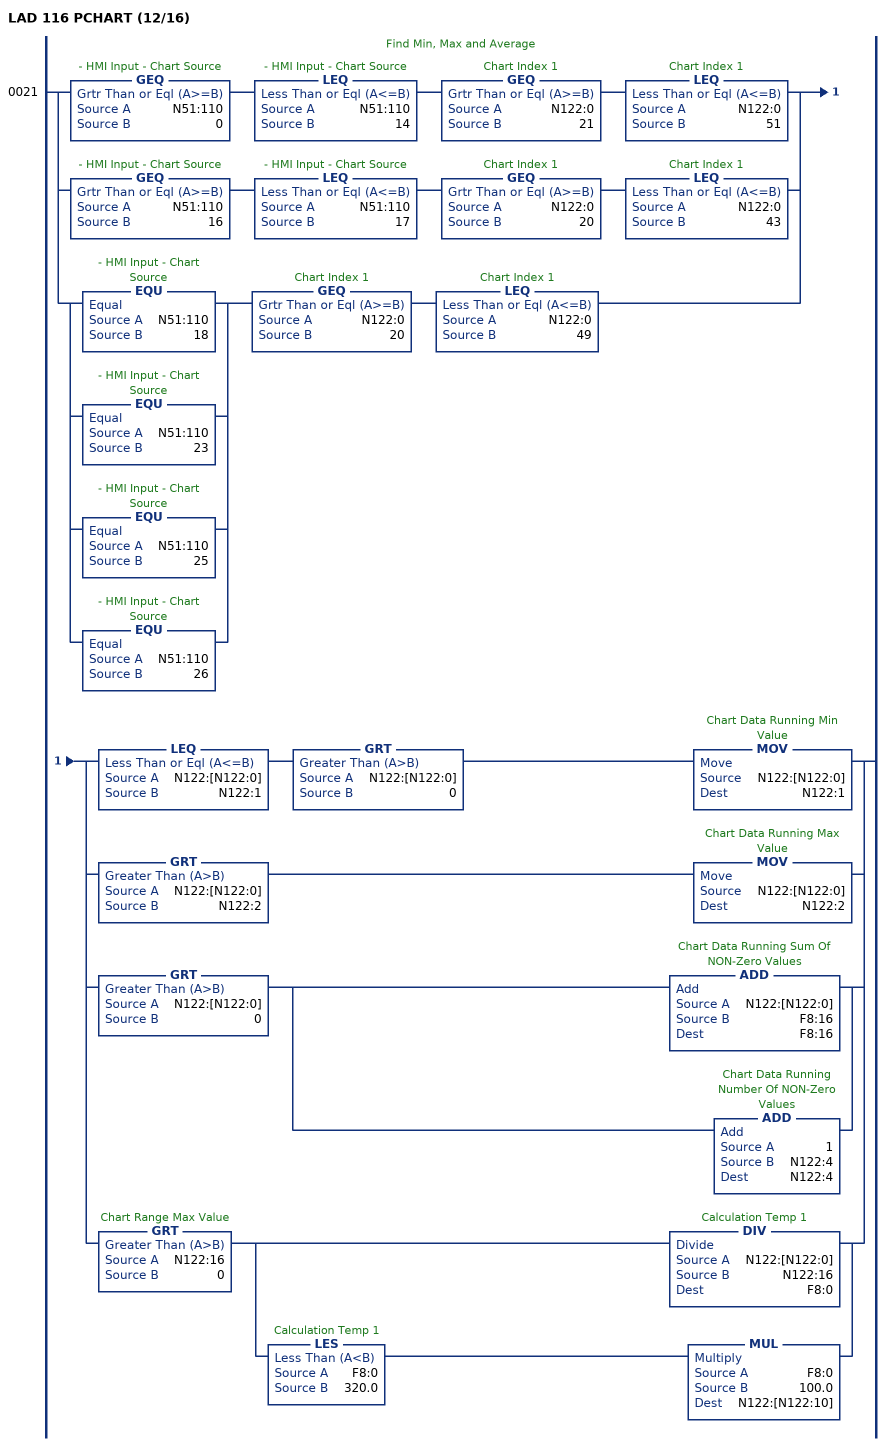
% Rung: 21 %
% Find Min, Max and Average %
SOR BST GEQ N51:110 0 LEQ N51:110 14 GEQ N122:0 21 LEQ N122:0 51 NXB GEQ N51:110 16 LEQ N51:110 17 GEQ N122:0 20 LEQ N122:0 43 NXB BST EQU N51:110 18 NXB EQU N51:110 23 NXB EQU N51:110 25 NXB EQU N51:110 26 BND GEQ N122:0 20 LEQ N122:0 49 BND BST LEQ N122:[N122:0] N122:1 GRT N122:[N122:0] 0 MOV N122:[N122:0] N122:1 NXB GRT N122:[N122:0] N122:2 MOV N122:[N122:0] N122:2 NXB GRT N122:[N122:0] 0 BST ADD N122:[N122:0] F8:16 F8:16 NXB ADD 1 N122:4 N122:4 BND NXB GRT N122:16 0 BST DIV N122:[N122:0] N122:16 F8:0 NXB LES F8:0 320.0 MUL F8:0 100.0 N122:[N122:10] BND BND EOR
%   N51:110  "- HMI Input - Chart Source" %
%   N122:0  "Chart Index 1" %
%   N122:1  "Chart Data Running Min Value" %
%   N122:2  "Chart Data Running Max Value" %
%   F8:16  "Chart Data Running Sum Of NON-Zero Values" %
%   N122:4  "Chart Data Running Number Of NON-Zero Values" %
%   N122:16  "Chart Range Max Value" %
%   F8:0  "Calculation Temp 1" %
%   N122:10  "Chart Index 2" %

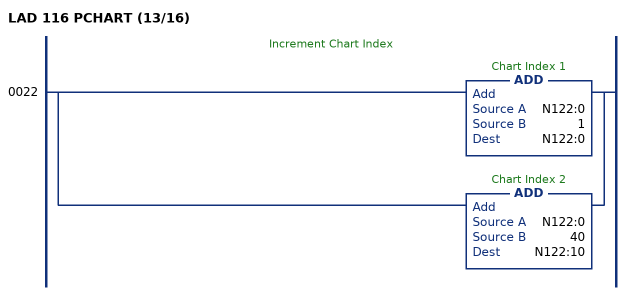
% Rung: 22 %
% Increment Chart Index %
SOR BST ADD N122:0 1 N122:0 NXB ADD N122:0 40 N122:10 BND EOR
%   N122:0  "Chart Index 1" %
%   N122:10  "Chart Index 2" %

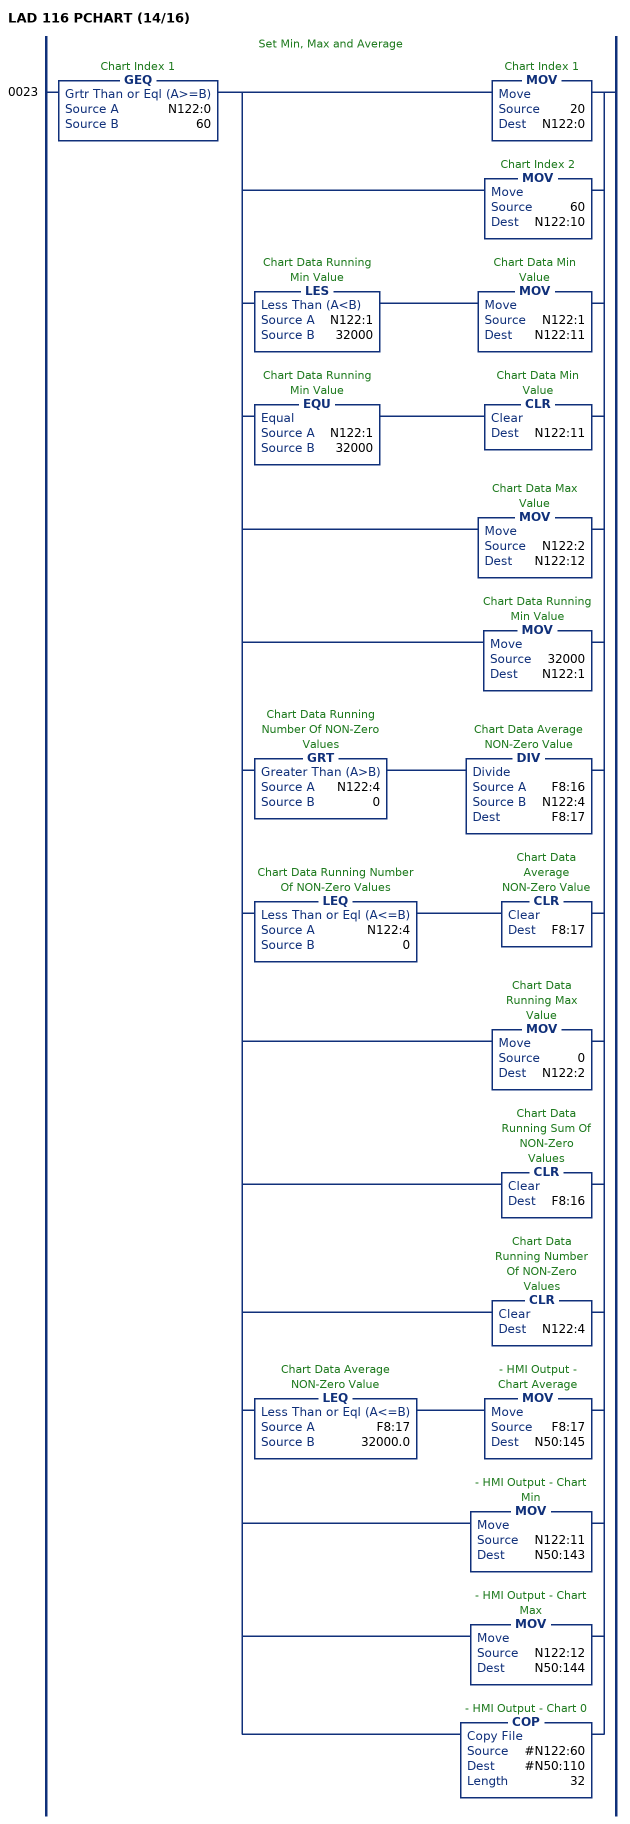
% Rung: 23 %
% Set Min, Max and Average %
SOR GEQ N122:0 60 BST MOV 20 N122:0 NXB MOV 60 N122:10 NXB BST LES N122:1 32000 MOV N122:1 N122:11 NXB EQU N122:1 32000 CLR N122:11 BND NXB MOV N122:2 N122:12 NXB MOV 32000 N122:1 NXB BST GRT N122:4 0 DIV F8:16 N122:4 F8:17 NXB LEQ N122:4 0 CLR F8:17 BND NXB MOV 0 N122:2 NXB CLR F8:16 NXB CLR N122:4 NXB LEQ F8:17 32000.0 MOV F8:17 N50:145 NXB MOV N122:11 N50:143 NXB MOV N122:12 N50:144 NXB COP #N122:60 #N50:110 32 BND EOR
%   N122:0  "Chart Index 1" %
%   N122:10  "Chart Index 2" %
%   N122:1  "Chart Data Running Min Value" %
%   N122:11  "Chart Data Min Value" %
%   N122:2  "Chart Data Running Max Value" %
%   N122:12  "Chart Data Max Value" %
%   N122:4  "Chart Data Running Number Of NON-Zero Values" %
%   F8:16  "Chart Data Running Sum Of NON-Zero Values" %
%   F8:17  "Chart Data Average NON-Zero Value" %
%   N50:145  "- HMI Output - Chart Average" %
%   N50:143  "- HMI Output - Chart Min" %
%   N50:144  "- HMI Output - Chart Max" %
%   N50:110  "- HMI Output - Chart 0" %

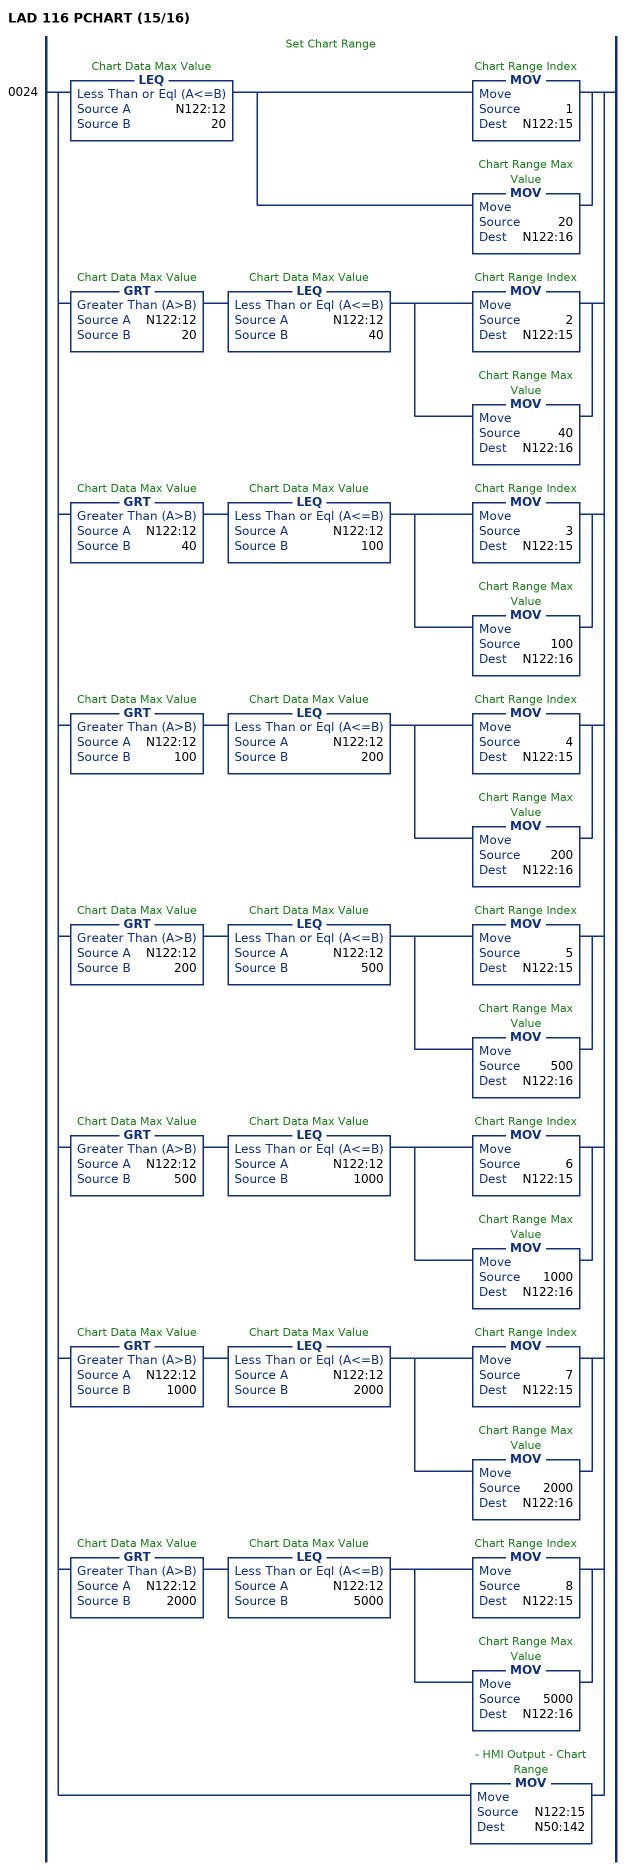
% Rung: 24 %
% Set Chart Range %
SOR BST LEQ N122:12 20 BST MOV 1 N122:15 NXB MOV 20 N122:16 BND NXB GRT N122:12 20 LEQ N122:12 40 BST MOV 2 N122:15 NXB MOV 40 N122:16 BND NXB GRT N122:12 40 LEQ N122:12 100 BST MOV 3 N122:15 NXB MOV 100 N122:16 BND NXB GRT N122:12 100 LEQ N122:12 200 BST MOV 4 N122:15 NXB MOV 200 N122:16 BND NXB GRT N122:12 200 LEQ N122:12 500 BST MOV 5 N122:15 NXB MOV 500 N122:16 BND NXB GRT N122:12 500 LEQ N122:12 1000 BST MOV 6 N122:15 NXB MOV 1000 N122:16 BND NXB GRT N122:12 1000 LEQ N122:12 2000 BST MOV 7 N122:15 NXB MOV 2000 N122:16 BND NXB GRT N122:12 2000 LEQ N122:12 5000 BST MOV 8 N122:15 NXB MOV 5000 N122:16 BND NXB MOV N122:15 N50:142 BND EOR
%   N122:12  "Chart Data Max Value" %
%   N122:15  "Chart Range Index" %
%   N122:16  "Chart Range Max Value" %
%   N50:142  "- HMI Output - Chart Range" %

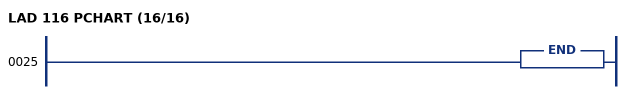
% Rung: 25 %
SOR END EOR

LADDER 117 "CDATA"    % Load Containment Data %
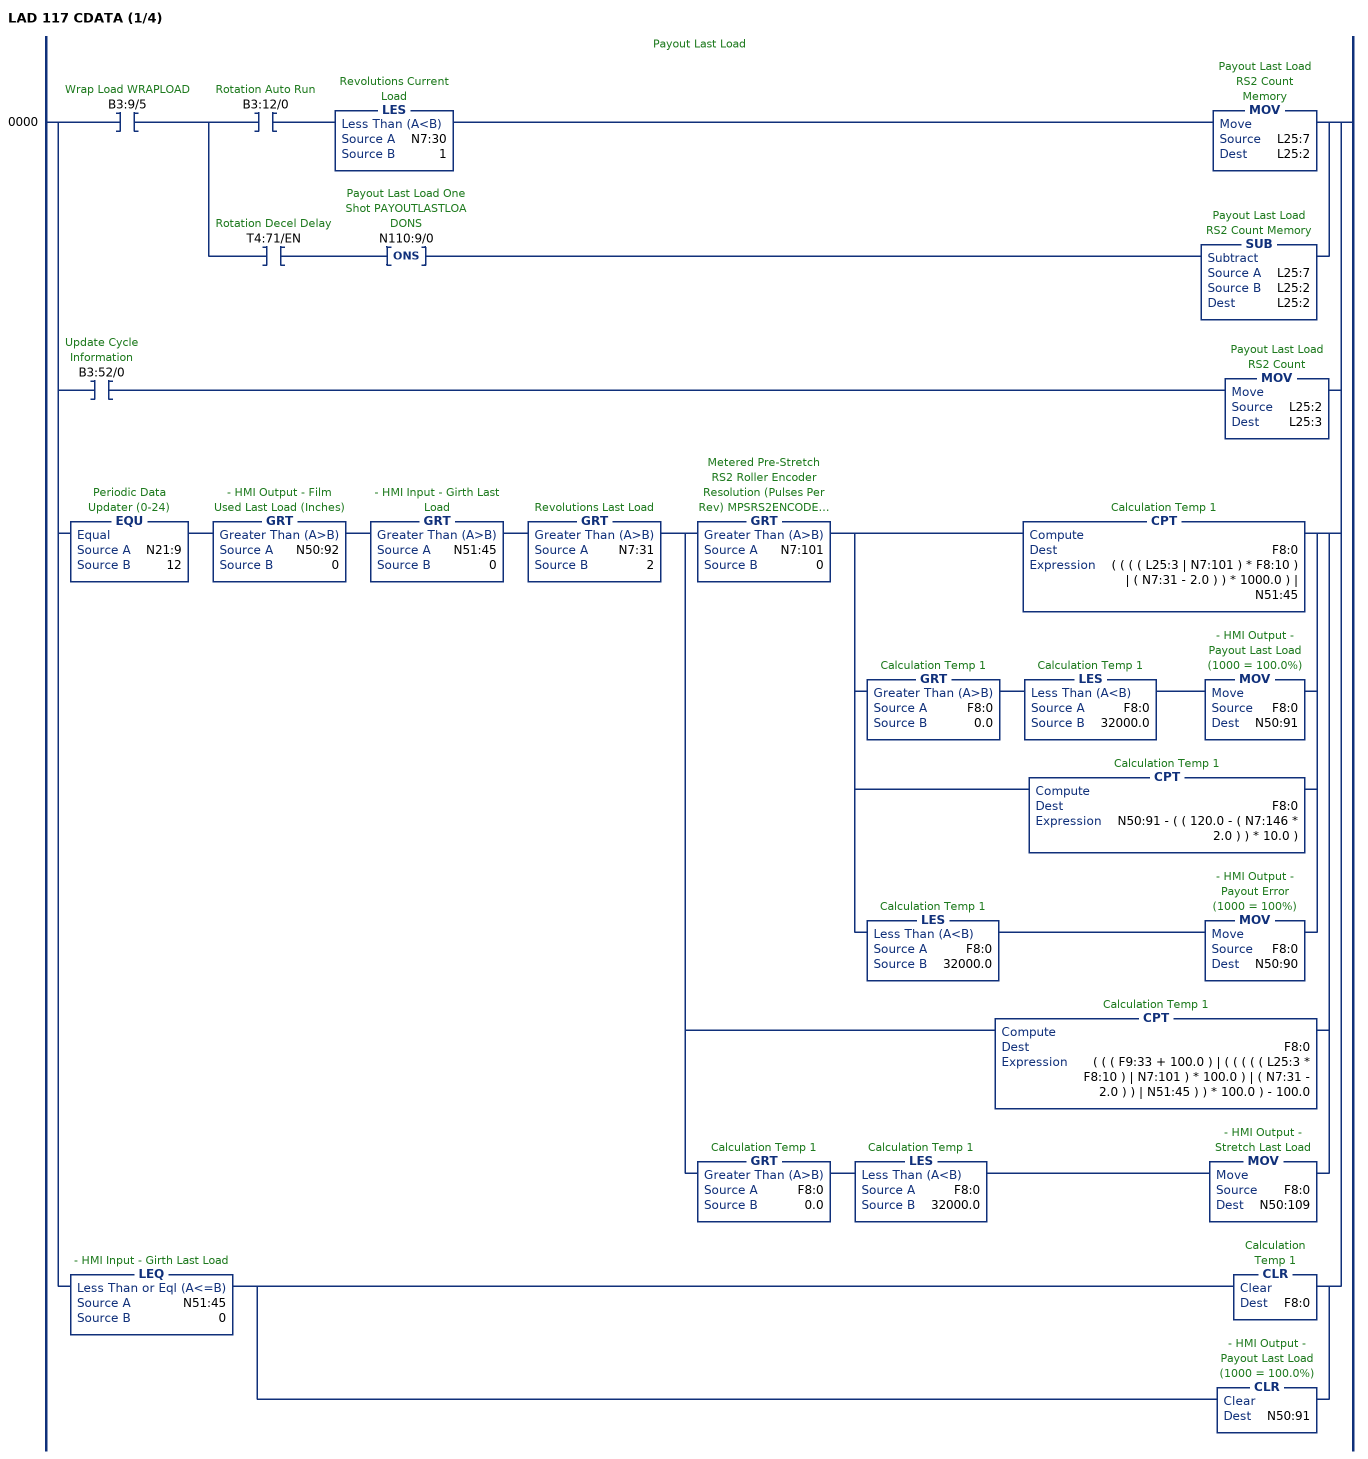
% Rung: 0 %
% Payout Last Load %
SOR BST XIC B3:9/5 BST XIC B3:12/0 LES N7:30 1 MOV L25:7 L25:2 NXB XIC T4:71/EN ONS N110:9/0 SUB L25:7 L25:2 L25:2 BND NXB XIC B3:52/0 MOV L25:2 L25:3 NXB EQU N21:9 12 GRT N50:92 0 GRT N51:45 0 GRT N7:31 2 BST GRT N7:101 0 BST CPT F8:0 " ( ( ( ( L25:3 | N7:101 ) * F8:10 ) | ( N7:31 - 2.0 ) ) * 1000.0 ) | N51:45 " NXB GRT F8:0 0.0 LES F8:0 32000.0 MOV F8:0 N50:91 NXB CPT F8:0 " N50:91 - ( ( 120.0 - ( N7:146 * 2.0 ) ) * 10.0 ) " NXB LES F8:0 32000.0 MOV F8:0 N50:90 BND NXB BST CPT F8:0 " ( ( ( F9:33 + 100.0 ) | ( ( ( ( ( L25:3 * F8:10 ) | N7:101 ) * 100.0 ) | ( N7:31 - 2.0 ) ) | N51:45 ) ) * 100.0 ) - 100.0 " NXB GRT F8:0 0.0 LES F8:0 32000.0 MOV F8:0 N50:109 BND BND NXB LEQ N51:45 0 BST CLR F8:0 NXB CLR N50:91 BND BND EOR
%   B3:9/5  WRAPLOAD  "Wrap Load" %
%   B3:12/0  "Rotation Auto Run" %
%   N7:30  "Revolutions Current Load" %
%   L25:7  "Metered Pre-Stretch RS2 Roller Current Count" %
%   L25:2  "Payout Last Load RS2 Count Memory" %
%   T4:71  "Rotation Decel Delay" %
%   N110:9/0  PAYOUTLASTLOADONS  "Payout Last Load One Shot" %
%   B3:52/0  "Update Cycle Information" %
%   L25:3  "Payout Last Load RS2 Count" %
%   N21:9  "Periodic Data Updater (0-24)" %
%   N50:92  "- HMI Output - Film Used Last Load (Inches)" %
%   N51:45  "- HMI Input - Girth Last Load" %
%   N7:31  "Revolutions Last Load" %
%   N7:101  MPSRS2ENCODERRES  "Metered Pre-Stretch RS2 Roller Encoder Resolution (Pulses Per Rev)" %
%   F8:0  "Calculation Temp 1" %
%   F8:10  MPSRS2CIRC  "Metered Pre-Stretch RS2 Roller Circumference (Inches)" %
%   N50:91  "- HMI Output - Payout Last Load (1000 = 100.0%)" %
%   N7:146  FORCELOADLAST  "Force At Load On Last Load" %
%   N50:90  "- HMI Output - Payout Error (1000 = 100%)" %
%   F9:33  PRESTRETCH  "Pre-Stretch %" %
%   N50:109  "- HMI Output - Stretch Last Load" %

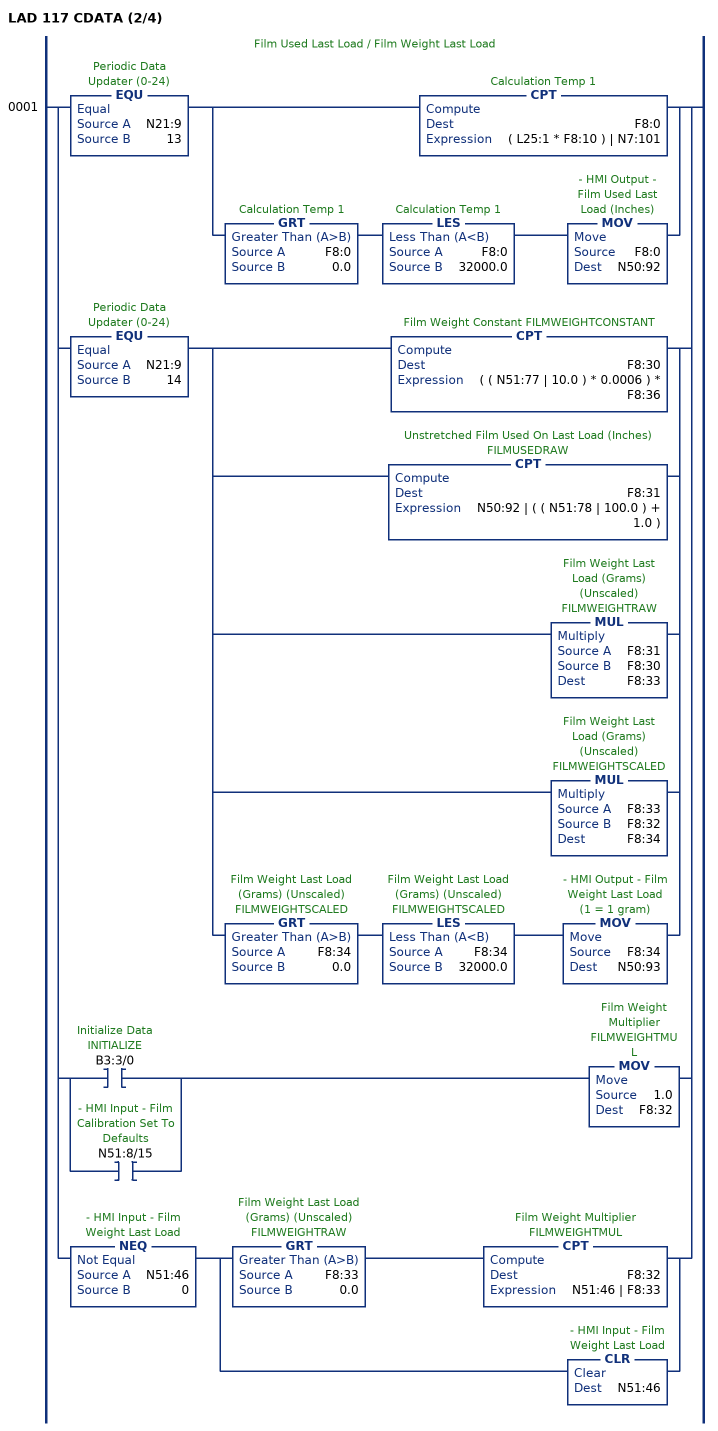
% Rung: 1 %
% Film Used Last Load / Film Weight Last Load %
SOR BST EQU N21:9 13 BST CPT F8:0 " ( L25:1 * F8:10 ) | N7:101 " NXB GRT F8:0 0.0 LES F8:0 32000.0 MOV F8:0 N50:92 BND NXB EQU N21:9 14 BST CPT F8:30 " ( ( N51:77 | 10.0 ) * 0.0006 ) * F8:36 " NXB CPT F8:31 " N50:92 | ( ( N51:78 | 100.0 ) + 1.0 ) " NXB BST MUL F8:31 F8:30 F8:33 NXB MUL F8:33 F8:32 F8:34 NXB GRT F8:34 0.0 LES F8:34 32000.0 MOV F8:34 N50:93 BND BND NXB BST XIC B3:3/0 NXB XIC N51:8/15 BND MOV 1.0 F8:32 NXB NEQ N51:46 0 BST GRT F8:33 0.0 CPT F8:32 " N51:46 | F8:33 " NXB CLR N51:46 BND BND EOR
%   N21:9  "Periodic Data Updater (0-24)" %
%   F8:0  "Calculation Temp 1" %
%   L25:1  "Metered Pre-Stretch RS2 Roller Counts Last Load" %
%   F8:10  MPSRS2CIRC  "Metered Pre-Stretch RS2 Roller Circumference (Inches)" %
%   N7:101  MPSRS2ENCODERRES  "Metered Pre-Stretch RS2 Roller Encoder Resolution (Pulses Per Rev)" %
%   N50:92  "- HMI Output - Film Used Last Load (Inches)" %
%   F8:30  FILMWEIGHTCONSTANT  "Film Weight Constant" %
%   N51:77  "- HMI Input - Preset Film Thickness (in microns)" %
%   F8:36  FILMSIZE  "Film Size (Inches)" %
%   F8:31  FILMUSEDRAW  "Unstretched Film Used On Last Load (Inches)" %
%   N51:78  "- HMI Input - Preset Prestretch %" %
%   F8:33  FILMWEIGHTRAW  "Film Weight Last Load (Grams) (Unscaled)" %
%   F8:32  FILMWEIGHTMUL  "Film Weight Multiplier" %
%   F8:34  FILMWEIGHTSCALED  "Film Weight Last Load (Grams) (Unscaled)" %
%   N50:93  "- HMI Output - Film Weight Last Load (1 = 1 gram)" %
%   B3:3/0  INITIALIZE  "Initialize Data" %
%   N51:8/15  "- HMI Input - Film Calibration Set To Defaults" %
%   N51:46  "- HMI Input - Film Weight Last Load" %

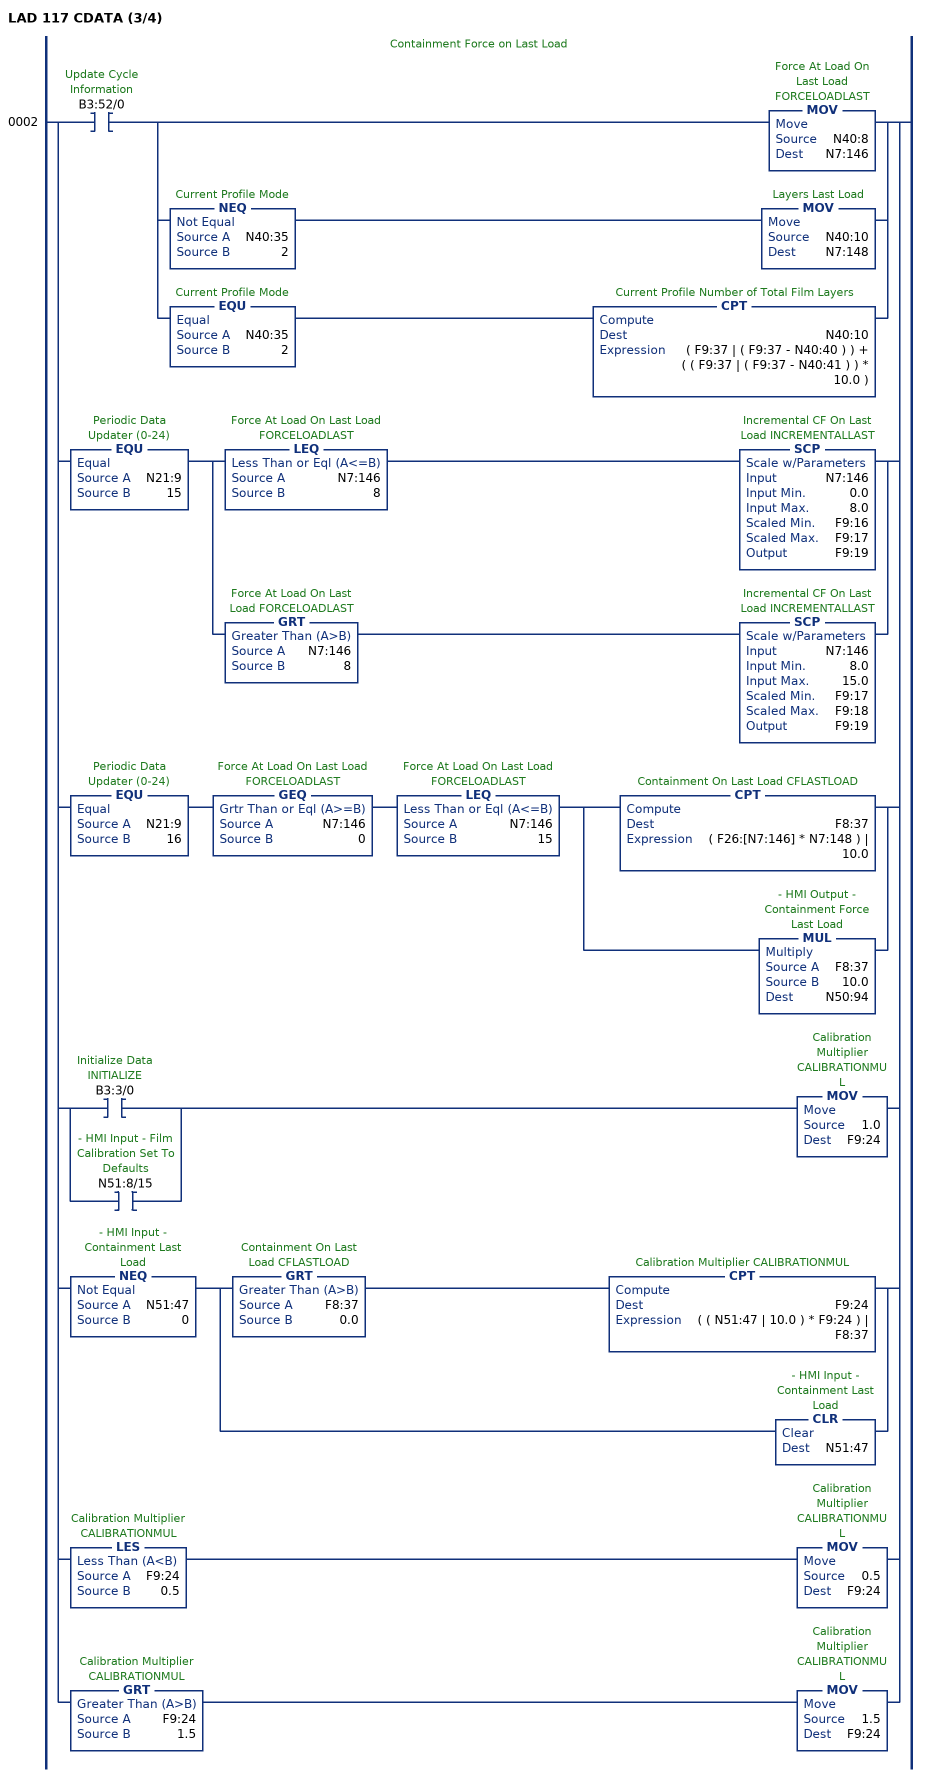
% Rung: 2 %
% Containment Force on Last Load %
SOR BST XIC B3:52/0 BST MOV N40:8 N7:146 NXB NEQ N40:35 2 MOV N40:10 N7:148 NXB EQU N40:35 2 CPT N40:10 " ( F9:37 | ( F9:37 - N40:40 ) ) + ( ( F9:37 | ( F9:37 - N40:41 ) ) * 10.0 ) " BND NXB EQU N21:9 15 BST LEQ N7:146 8 SCP N7:146 0.0 8.0 F9:16 F9:17 F9:19 NXB GRT N7:146 8 SCP N7:146 8.0 15.0 F9:17 F9:18 F9:19 BND NXB EQU N21:9 16 GEQ N7:146 0 LEQ N7:146 15 BST CPT F8:37 " ( F26:[N7:146] * N7:148 ) | 10.0 " NXB MUL F8:37 10.0 N50:94 BND NXB BST XIC B3:3/0 NXB XIC N51:8/15 BND MOV 1.0 F9:24 NXB NEQ N51:47 0 BST GRT F8:37 0.0 CPT F9:24 " ( ( N51:47 | 10.0 ) * F9:24 ) | F8:37 " NXB CLR N51:47 BND NXB LES F9:24 0.5 MOV 0.5 F9:24 NXB GRT F9:24 1.5 MOV 1.5 F9:24 BND EOR
%   B3:52/0  "Update Cycle Information" %
%   N40:8  "Current Profile Force At Load" %
%   N7:146  FORCELOADLAST  "Force At Load On Last Load" %
%   N40:35  "Current Profile Mode" %
%   N40:10  "Current Profile Number of Total Film Layers" %
%   N7:148  "Layers Last Load" %
%   F9:37  "Film Width Scaled for Film Tension" %
%   N21:9  "Periodic Data Updater (0-24)" %
%   F9:16  INCREMENTALAT0  "Incremental CF At WF0 For A Given Film Thickness" %
%   F9:17  INCREMENTALAT8  "Incremental CF At WF8 For A Given Film Thickness" %
%   F9:19  INCREMENTALLAST  "Incremental CF On Last Load" %
%   F9:18  INCREMENTALAT15  "Incremental CF At WF15 For A Given Film Thickness" %
%   F8:37  CFLASTLOAD  "Containment On Last Load" %
%   N50:94  "- HMI Output - Containment Force Last Load" %
%   B3:3/0  INITIALIZE  "Initialize Data" %
%   N51:8/15  "- HMI Input - Film Calibration Set To Defaults" %
%   F9:24  CALIBRATIONMUL  "Calibration Multiplier" %
%   N51:47  "- HMI Input - Containment Last Load" %

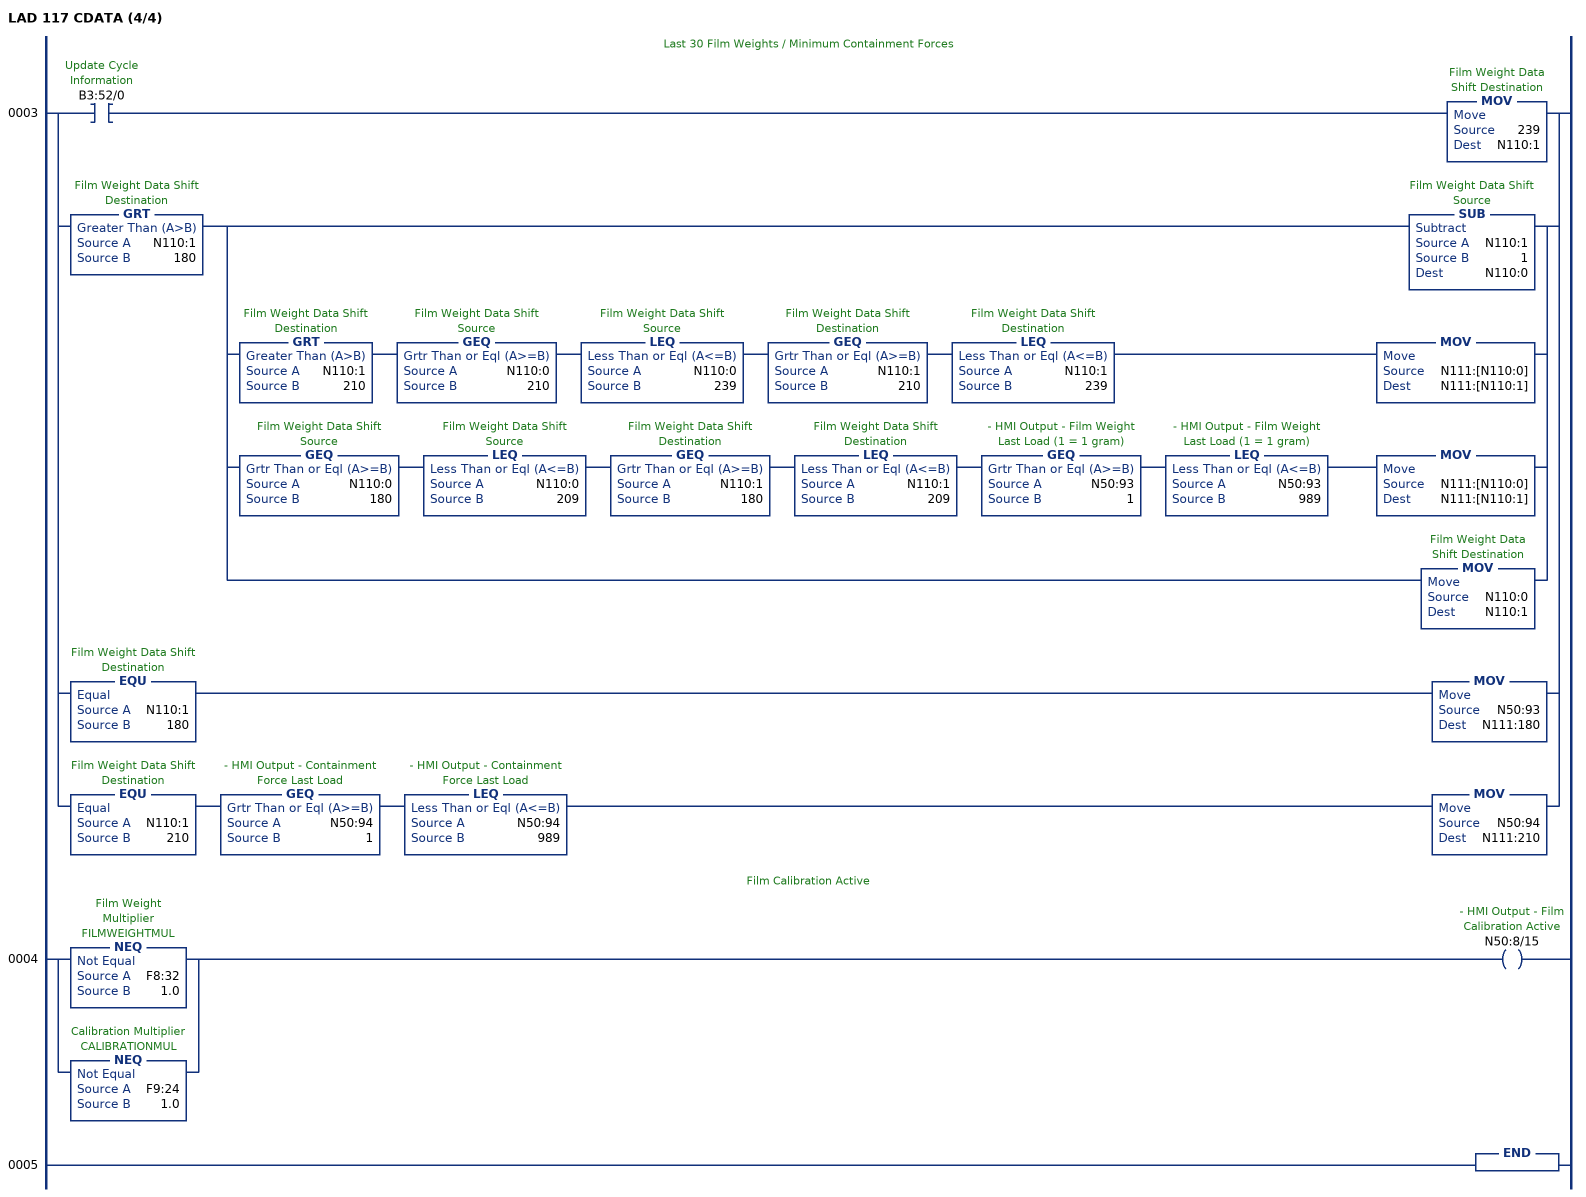
% Rung: 3 %
% Last 30 Film Weights / Minimum Containment Forces %
SOR BST XIC B3:52/0 MOV 239 N110:1 NXB GRT N110:1 180 BST SUB N110:1 1 N110:0 NXB GRT N110:1 210 GEQ N110:0 210 LEQ N110:0 239 GEQ N110:1 210 LEQ N110:1 239 MOV N111:[N110:0] N111:[N110:1] NXB GEQ N110:0 180 LEQ N110:0 209 GEQ N110:1 180 LEQ N110:1 209 GEQ N50:93 1 LEQ N50:93 989 MOV N111:[N110:0] N111:[N110:1] NXB MOV N110:0 N110:1 BND NXB EQU N110:1 180 MOV N50:93 N111:180 NXB EQU N110:1 210 GEQ N50:94 1 LEQ N50:94 989 MOV N50:94 N111:210 BND EOR
%   B3:52/0  "Update Cycle Information" %
%   N110:1  "Film Weight Data Shift Destination" %
%   N110:0  "Film Weight Data Shift Source" %
%   N50:93  "- HMI Output - Film Weight Last Load (1 = 1 gram)" %
%   N50:94  "- HMI Output - Containment Force Last Load" %
% Rung: 4 %
% Film Calibration Active %
SOR BST NEQ F8:32 1.0 NXB NEQ F9:24 1.0 BND OTE N50:8/15 EOR
%   F8:32  FILMWEIGHTMUL  "Film Weight Multiplier" %
%   F9:24  CALIBRATIONMUL  "Calibration Multiplier" %
%   N50:8/15  "- HMI Output - Film Calibration Active" %
% Rung: 5 %
SOR END EOR

LADDER 214 "MPS CALC"
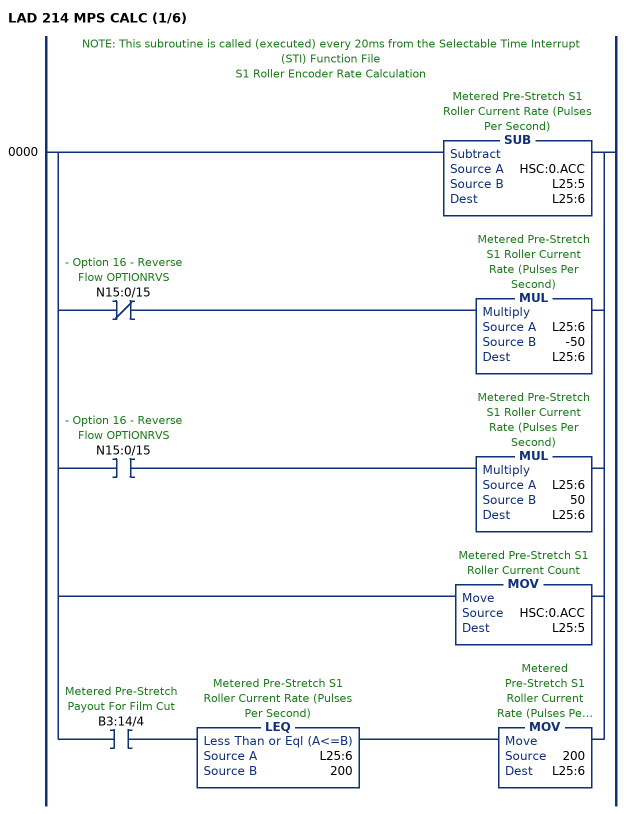
% Rung: 0 %
% NOTE: This subroutine is called (executed) every 20ms from the Selectable Time Interrupt (STI) Function File
% 
% S1 Roller Encoder Rate Calculation %
SOR BST SUB HSC:0.ACC L25:5 L25:6 NXB XIO N15:0/15 MUL L25:6 -50 L25:6 NXB XIC N15:0/15 MUL L25:6 50 L25:6 NXB MOV HSC:0.ACC L25:5 NXB XIC B3:14/4 LEQ L25:6 200 MOV 200 L25:6 BND EOR
%   L25:5  "Metered Pre-Stretch S1 Roller Current Count" %
%   L25:6  "Metered Pre-Stretch S1 Roller Current Rate (Pulses Per Second)" %
%   N15:0/15  OPTIONRVS  "- Option 16 - Reverse Flow" %
%   B3:14/4  "Metered Pre-Stretch Payout For Film Cut" %

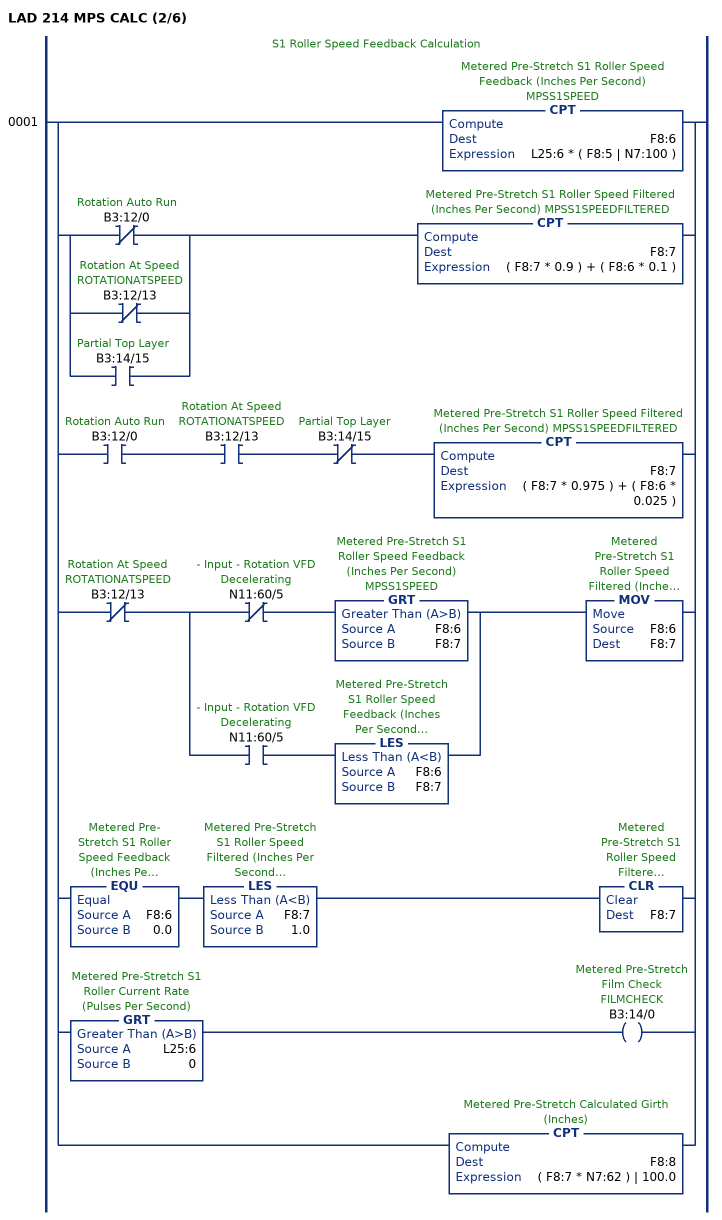
% Rung: 1 %
% S1 Roller Speed Feedback Calculation %
SOR BST CPT F8:6 " L25:6 * ( F8:5 | N7:100 ) " NXB BST XIO B3:12/0 NXB XIO B3:12/13 NXB XIC B3:14/15 BND CPT F8:7 " ( F8:7 * 0.9 ) + ( F8:6 * 0.1 ) " NXB XIC B3:12/0 XIC B3:12/13 XIO B3:14/15 CPT F8:7 " ( F8:7 * 0.975 ) + ( F8:6 * 0.025 ) " NXB XIO B3:12/13 BST XIO N11:60/5 GRT F8:6 F8:7 NXB XIC N11:60/5 LES F8:6 F8:7 BND MOV F8:6 F8:7 NXB EQU F8:6 0.0 LES F8:7 1.0 CLR F8:7 NXB GRT L25:6 0 OTE B3:14/0 NXB CPT F8:8 " ( F8:7 * N7:62 ) | 100.0 " BND EOR
%   F8:6  MPSS1SPEED  "Metered Pre-Stretch S1 Roller Speed Feedback (Inches Per Second)" %
%   L25:6  "Metered Pre-Stretch S1 Roller Current Rate (Pulses Per Second)" %
%   F8:5  MPSS1CIRC  "Metered Pre-Stretch S1 Roller Circumference (Inches)" %
%   N7:100  MPSS1ENCODERRES  "Metered Pre-Stretch S1 Roller Encoder Resolution (Pulses Per Rev)" %
%   B3:12/0  "Rotation Auto Run" %
%   B3:12/13  ROTATIONATSPEED  "Rotation At Speed" %
%   B3:14/15  "Partial Top Layer" %
%   F8:7  MPSS1SPEEDFILTERED  "Metered Pre-Stretch S1 Roller Speed Filtered (Inches Per Second)" %
%   N11:60/5  "- Input - Rotation VFD Decelerating" %
%   B3:14/0  FILMCHECK  "Metered Pre-Stretch Film Check" %
%   F8:8  "Metered Pre-Stretch Calculated Girth (Inches)" %
%   N7:62  "Rotation Revolution Time (100 = 1.00s)" %

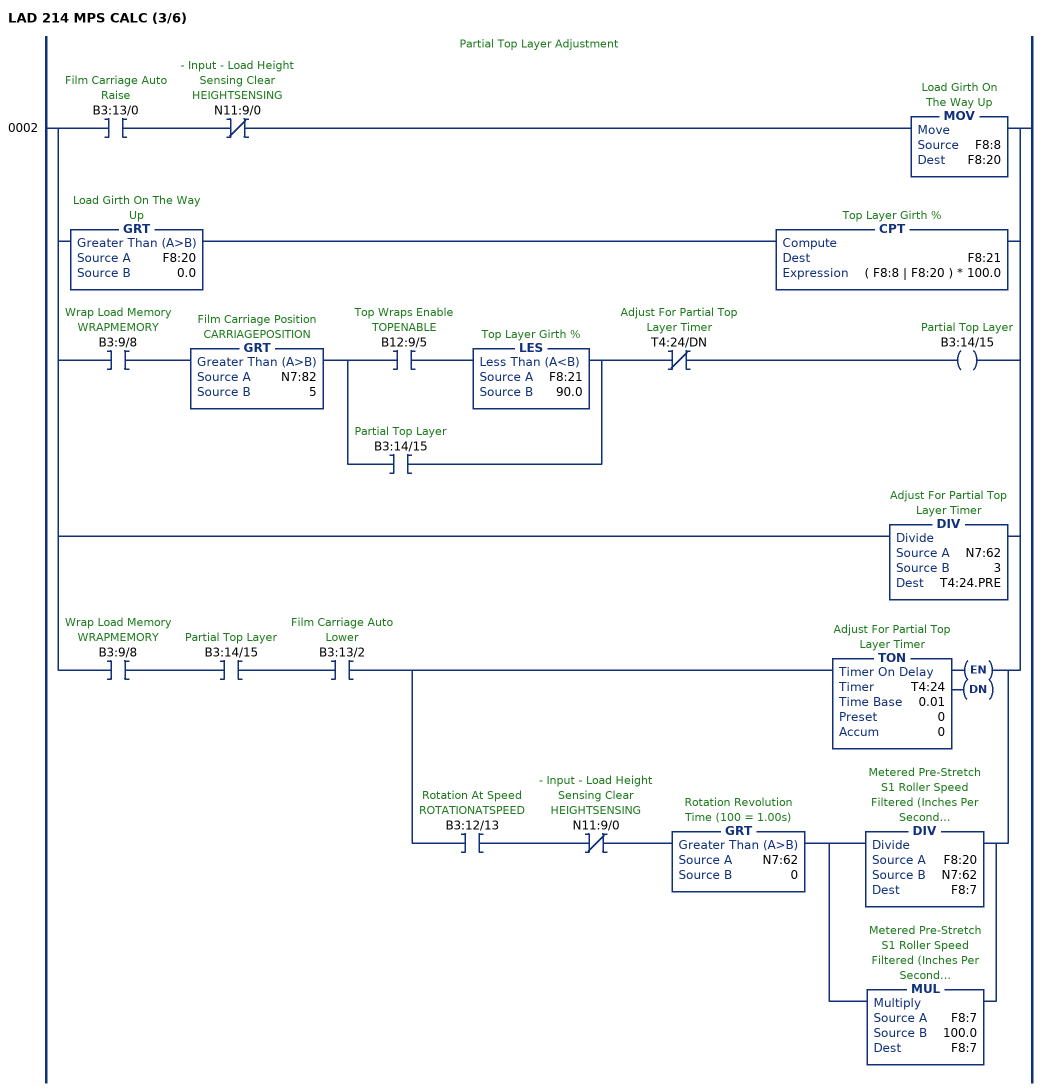
% Rung: 2 %
% Partial Top Layer Adjustment %
SOR BST XIC B3:13/0 XIO N11:9/0 MOV F8:8 F8:20 NXB GRT F8:20 0.0 CPT F8:21 " ( F8:8 | F8:20 ) * 100.0 " NXB XIC B3:9/8 GRT N7:82 5 BST XIC B12:9/5 LES F8:21 90.0 NXB XIC B3:14/15 BND XIO T4:24/DN OTE B3:14/15 NXB DIV N7:62 3 T4:24.PRE NXB XIC B3:9/8 XIC B3:14/15 XIC B3:13/2 BST TON T4:24 0.01 0 0 NXB XIC B3:12/13 XIO N11:9/0 GRT N7:62 0 BST DIV F8:20 N7:62 F8:7 NXB MUL F8:7 100.0 F8:7 BND BND BND EOR
%   B3:13/0  "Film Carriage Auto Raise" %
%   N11:9/0  HEIGHTSENSING  "- Input - Load Height Sensing Clear" %
%   F8:8  "Metered Pre-Stretch Calculated Girth (Inches)" %
%   F8:20  "Load Girth On The Way Up" %
%   F8:21  "Top Layer Girth %" %
%   B3:9/8  WRAPMEMORY  "Wrap Load Memory" %
%   N7:82  CARRIAGEPOSITION  "Film Carriage Position" %
%   B12:9/5  TOPENABLE  "Top Wraps Enable" %
%   B3:14/15  "Partial Top Layer" %
%   T4:24  "Adjust For Partial Top Layer Timer" %
%   N7:62  "Rotation Revolution Time (100 = 1.00s)" %
%   B3:13/2  "Film Carriage Auto Lower" %
%   B3:12/13  ROTATIONATSPEED  "Rotation At Speed" %
%   F8:7  MPSS1SPEEDFILTERED  "Metered Pre-Stretch S1 Roller Speed Filtered (Inches Per Second)" %

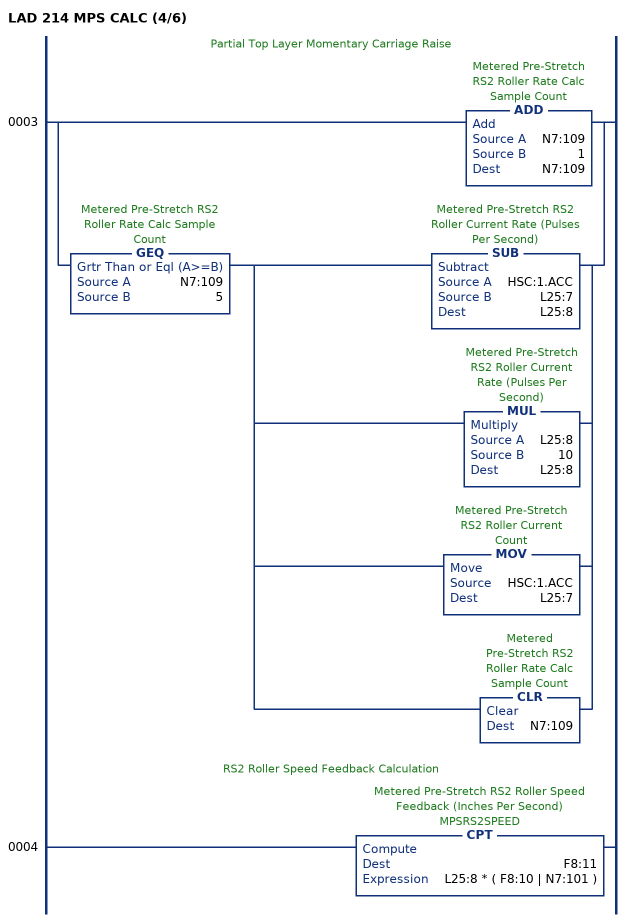
% Rung: 3 %
% Partial Top Layer Momentary Carriage Raise %
SOR BST ADD N7:109 1 N7:109 NXB GEQ N7:109 5 BST SUB HSC:1.ACC L25:7 L25:8 NXB MUL L25:8 10 L25:8 NXB MOV HSC:1.ACC L25:7 NXB CLR N7:109 BND BND EOR
%   N7:109  "Metered Pre-Stretch RS2 Roller Rate Calc Sample Count" %
%   L25:7  "Metered Pre-Stretch RS2 Roller Current Count" %
%   L25:8  "Metered Pre-Stretch RS2 Roller Current Rate (Pulses Per Second)" %
% Rung: 4 %
% RS2 Roller Speed Feedback Calculation %
SOR CPT F8:11 " L25:8 * ( F8:10 | N7:101 ) " EOR
%   F8:11  MPSRS2SPEED  "Metered Pre-Stretch RS2 Roller Speed Feedback (Inches Per Second)" %
%   L25:8  "Metered Pre-Stretch RS2 Roller Current Rate (Pulses Per Second)" %
%   F8:10  MPSRS2CIRC  "Metered Pre-Stretch RS2 Roller Circumference (Inches)" %
%   N7:101  MPSRS2ENCODERRES  "Metered Pre-Stretch RS2 Roller Encoder Resolution (Pulses Per Rev)" %

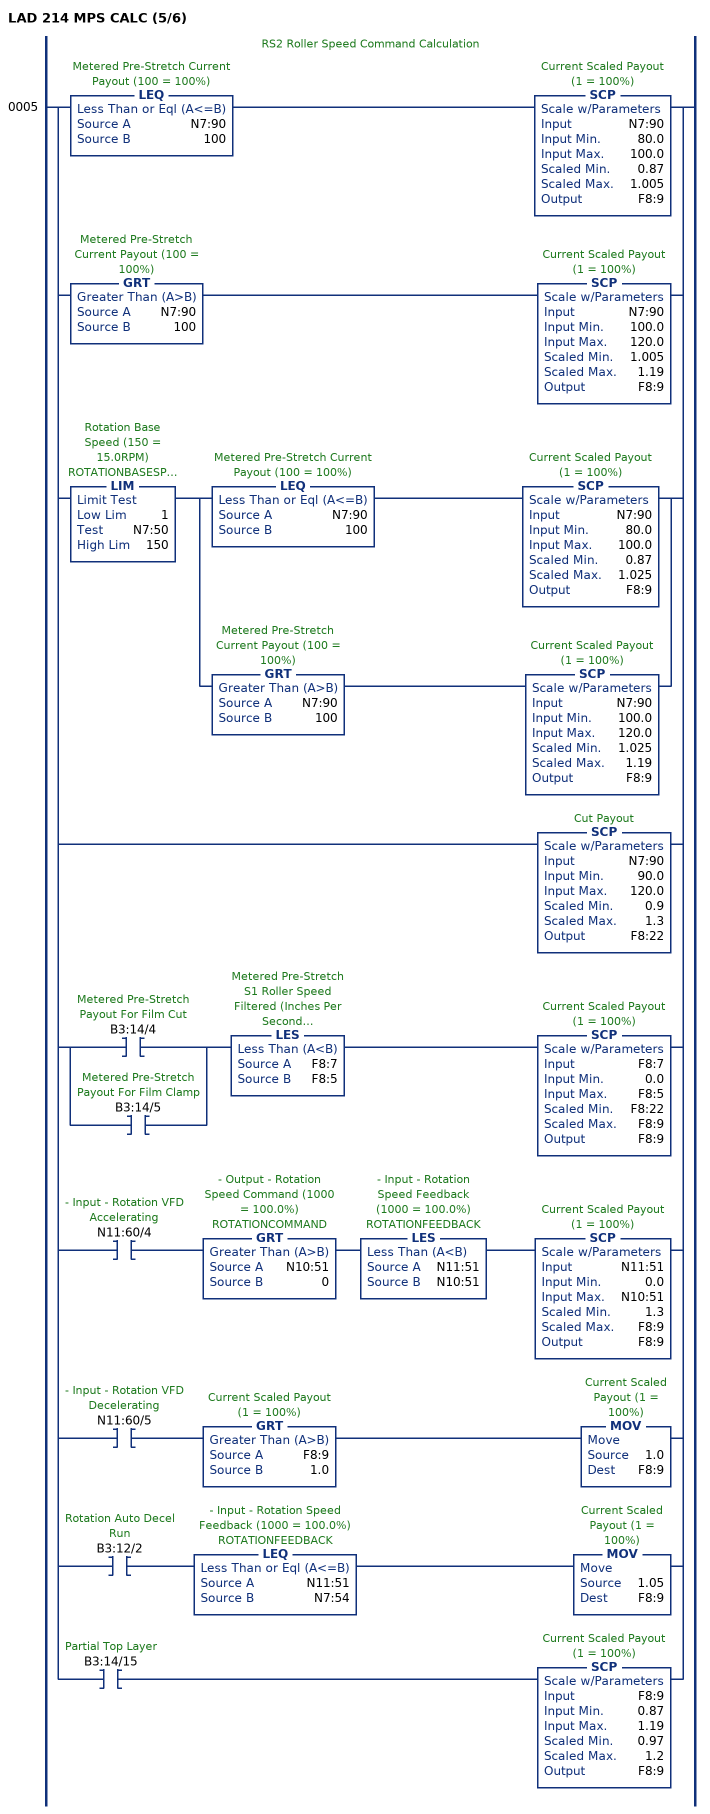
% Rung: 5 %
% RS2 Roller Speed Command Calculation %
SOR BST BST LEQ N7:90 100 SCP N7:90 80.0 100.0 0.87 1.005 F8:9 NXB GRT N7:90 100 SCP N7:90 100.0 120.0 1.005 1.19 F8:9 NXB LIM 1 N7:50 150 BST LEQ N7:90 100 SCP N7:90 80.0 100.0 0.87 1.025 F8:9 NXB GRT N7:90 100 SCP N7:90 100.0 120.0 1.025 1.19 F8:9 BND NXB SCP N7:90 90.0 120.0 0.9 1.3 F8:22 BND NXB BST XIC B3:14/4 NXB XIC B3:14/5 BND LES F8:7 F8:5 SCP F8:7 0.0 F8:5 F8:22 F8:9 F8:9 NXB XIC N11:60/4 GRT N10:51 0 LES N11:51 N10:51 SCP N11:51 0.0 N10:51 1.3 F8:9 F8:9 NXB XIC N11:60/5 GRT F8:9 1.0 MOV 1.0 F8:9 NXB XIC B3:12/2 LEQ N11:51 N7:54 MOV 1.05 F8:9 NXB XIC B3:14/15 SCP F8:9 0.87 1.19 0.97 1.2 F8:9 BND EOR
%   N7:90  "Metered Pre-Stretch Current Payout (100 = 100%)" %
%   F8:9  "Current Scaled Payout (1 = 100%)" %
%   N7:50  ROTATIONBASESPEED  "Rotation Base Speed (150 = 15.0RPM)" %
%   F8:22  "Cut Payout" %
%   B3:14/4  "Metered Pre-Stretch Payout For Film Cut" %
%   B3:14/5  "Metered Pre-Stretch Payout For Film Clamp" %
%   F8:7  MPSS1SPEEDFILTERED  "Metered Pre-Stretch S1 Roller Speed Filtered (Inches Per Second)" %
%   F8:5  MPSS1CIRC  "Metered Pre-Stretch S1 Roller Circumference (Inches)" %
%   N11:60/4  "- Input - Rotation VFD Accelerating" %
%   N10:51  ROTATIONCOMMAND  "- Output - Rotation Speed Command (1000 = 100.0%)" %
%   N11:51  ROTATIONFEEDBACK  "- Input - Rotation Speed Feedback (1000 = 100.0%)" %
%   N11:60/5  "- Input - Rotation VFD Decelerating" %
%   B3:12/2  "Rotation Auto Decel Run" %
%   N7:54  "Rotation Home Speed (1000 = 100.0%)" %
%   B3:14/15  "Partial Top Layer" %

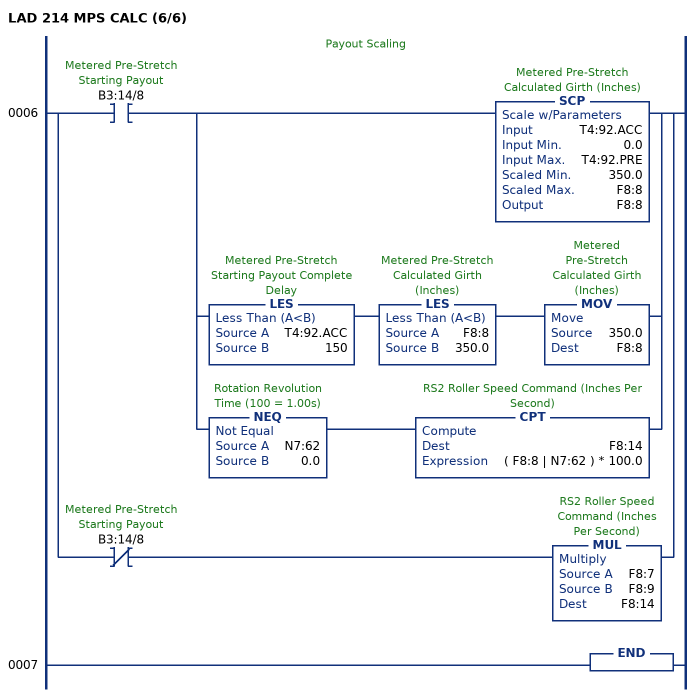
% Rung: 6 %
% Payout Scaling %
SOR BST XIC B3:14/8 BST SCP T4:92.ACC 0.0 T4:92.PRE 350.0 F8:8 F8:8 NXB LES T4:92.ACC 150 LES F8:8 350.0 MOV 350.0 F8:8 NXB NEQ N7:62 0.0 CPT F8:14 " ( F8:8 | N7:62 ) * 100.0 " BND NXB XIO B3:14/8 MUL F8:7 F8:9 F8:14 BND EOR
%   B3:14/8  "Metered Pre-Stretch Starting Payout" %
%   T4:92  "Metered Pre-Stretch Starting Payout Complete Delay" %
%   F8:8  "Metered Pre-Stretch Calculated Girth (Inches)" %
%   N7:62  "Rotation Revolution Time (100 = 1.00s)" %
%   F8:14  "RS2 Roller Speed Command (Inches Per Second)" %
%   F8:7  MPSS1SPEEDFILTERED  "Metered Pre-Stretch S1 Roller Speed Filtered (Inches Per Second)" %
%   F8:9  "Current Scaled Payout (1 = 100%)" %
% Rung: 7 %
SOR END EOR

LADDER 250 "VFD MODBUS"
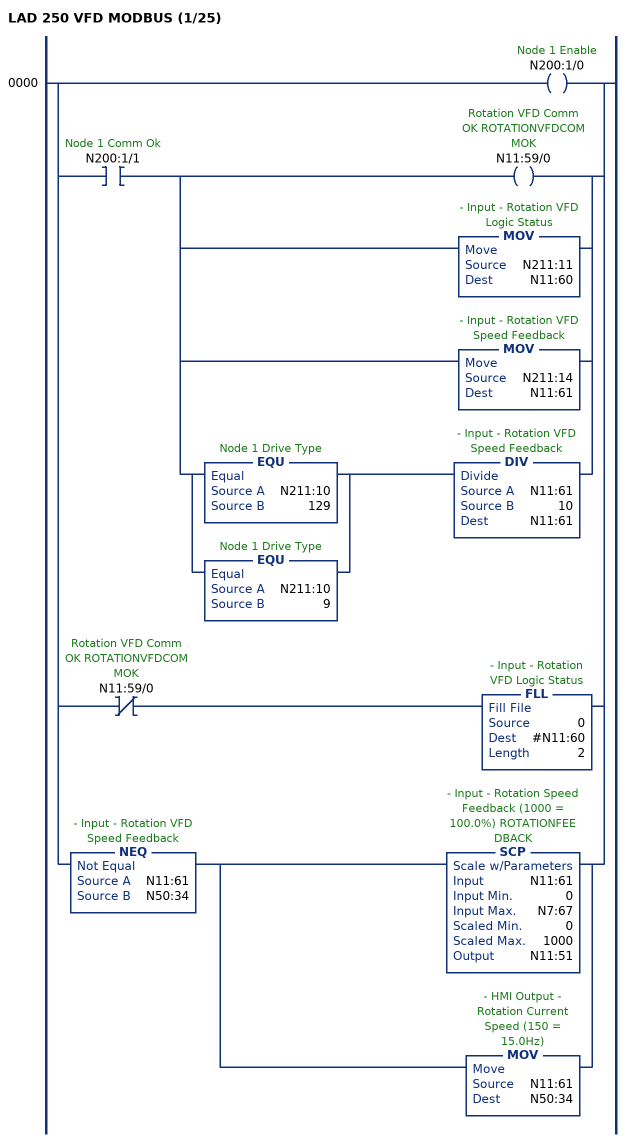
% Rung: 0 %
SOR BST OTE N200:1/0 NXB XIC N200:1/1 BST OTE N11:59/0 NXB MOV N211:11 N11:60 NXB MOV N211:14 N11:61 NXB BST EQU N211:10 129 NXB EQU N211:10 9 BND DIV N11:61 10 N11:61 BND NXB XIO N11:59/0 FLL 0 #N11:60 2 NXB NEQ N11:61 N50:34 BST SCP N11:61 0 N7:67 0 1000 N11:51 NXB MOV N11:61 N50:34 BND BND EOR
%   N200:1/0  "Node 1 Enable" %
%   N200:1/1  "Node 1 Comm Ok" %
%   N11:59/0  ROTATIONVFDCOMMOK  "Rotation VFD Comm OK" %
%   N211:11  "Node 1 Logic Status" %
%   N11:60  "- Input - Rotation VFD Logic Status" %
%   N211:14  "Node 1 Speed Feedback" %
%   N11:61  "- Input - Rotation VFD Speed Feedback" %
%   N211:10  "Node 1 Drive Type" %
%   N50:34  "- HMI Output - Rotation Current Speed (150 = 15.0Hz)" %
%   N7:67  "Rotation VFD Max Hz (150 = 15.0Hz)" %
%   N11:51  ROTATIONFEEDBACK  "- Input - Rotation Speed Feedback (1000 = 100.0%)" %

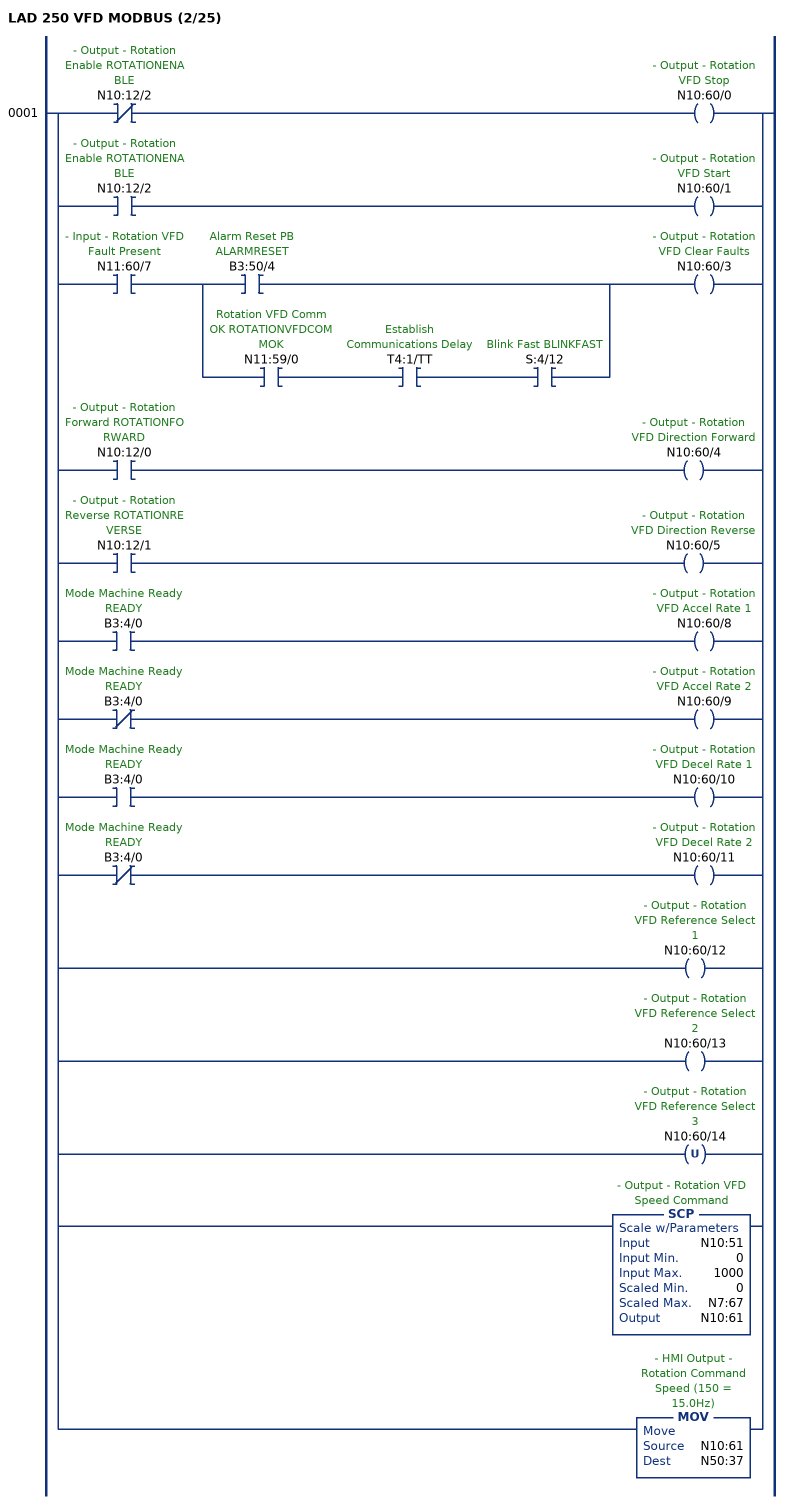
% Rung: 1 %
SOR BST XIO N10:12/2 OTE N10:60/0 NXB XIC N10:12/2 OTE N10:60/1 NXB XIC N11:60/7 BST XIC B3:50/4 NXB XIC N11:59/0 XIC T4:1/TT XIC S:4/12 BND OTE N10:60/3 NXB XIC N10:12/0 OTE N10:60/4 NXB XIC N10:12/1 OTE N10:60/5 NXB XIC B3:4/0 OTE N10:60/8 NXB XIO B3:4/0 OTE N10:60/9 NXB XIC B3:4/0 OTE N10:60/10 NXB XIO B3:4/0 OTE N10:60/11 NXB OTE N10:60/12 NXB OTE N10:60/13 NXB OTU N10:60/14 NXB SCP N10:51 0 1000 0 N7:67 N10:61 NXB MOV N10:61 N50:37 BND EOR
%   N10:12/2  ROTATIONENABLE  "- Output - Rotation Enable" %
%   N10:60/0  "- Output - Rotation VFD Stop" %
%   N10:60/1  "- Output - Rotation VFD Start" %
%   N11:60/7  "- Input - Rotation VFD Fault Present" %
%   B3:50/4  ALARMRESET  "Alarm Reset PB" %
%   N11:59/0  ROTATIONVFDCOMMOK  "Rotation VFD Comm OK" %
%   T4:1  "Establish Communications Delay" %
%   S:4/12  BLINKFAST  "Blink Fast" %
%   N10:60/3  "- Output - Rotation VFD Clear Faults" %
%   N10:12/0  ROTATIONFORWARD  "- Output - Rotation Forward" %
%   N10:60/4  "- Output - Rotation VFD Direction Forward" %
%   N10:12/1  ROTATIONREVERSE  "- Output - Rotation Reverse" %
%   N10:60/5  "- Output - Rotation VFD Direction Reverse" %
%   B3:4/0  READY  "Mode Machine Ready" %
%   N10:60/8  "- Output - Rotation VFD Accel Rate 1" %
%   N10:60/9  "- Output - Rotation VFD Accel Rate 2" %
%   N10:60/10  "- Output - Rotation VFD Decel Rate 1" %
%   N10:60/11  "- Output - Rotation VFD Decel Rate 2" %
%   N10:60/12  "- Output - Rotation VFD Reference Select 1" %
%   N10:60/13  "- Output - Rotation VFD Reference Select 2" %
%   N10:60/14  "- Output - Rotation VFD Reference Select 3" %
%   N10:51  ROTATIONCOMMAND  "- Output - Rotation Speed Command (1000 = 100.0%)" %
%   N7:67  "Rotation VFD Max Hz (150 = 15.0Hz)" %
%   N10:61  "- Output - Rotation VFD Speed Command" %
%   N50:37  "- HMI Output - Rotation Command Speed (150 = 15.0Hz)" %

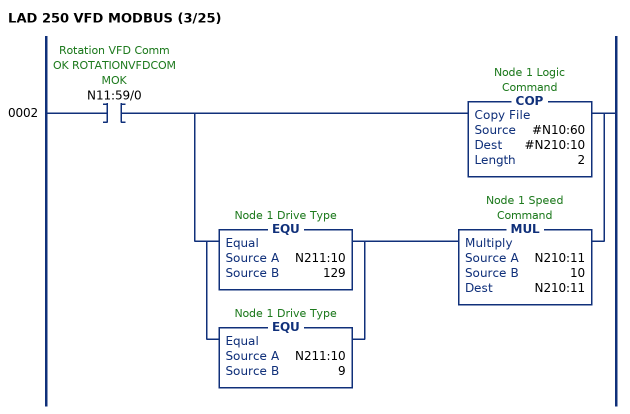
% Rung: 2 %
SOR XIC N11:59/0 BST COP #N10:60 #N210:10 2 NXB BST EQU N211:10 129 NXB EQU N211:10 9 BND MUL N210:11 10 N210:11 BND EOR
%   N11:59/0  ROTATIONVFDCOMMOK  "Rotation VFD Comm OK" %
%   N10:60  "- Output - Rotation VFD Logic Command" %
%   N210:10  "Node 1 Logic Command" %
%   N211:10  "Node 1 Drive Type" %
%   N210:11  "Node 1 Speed Command" %

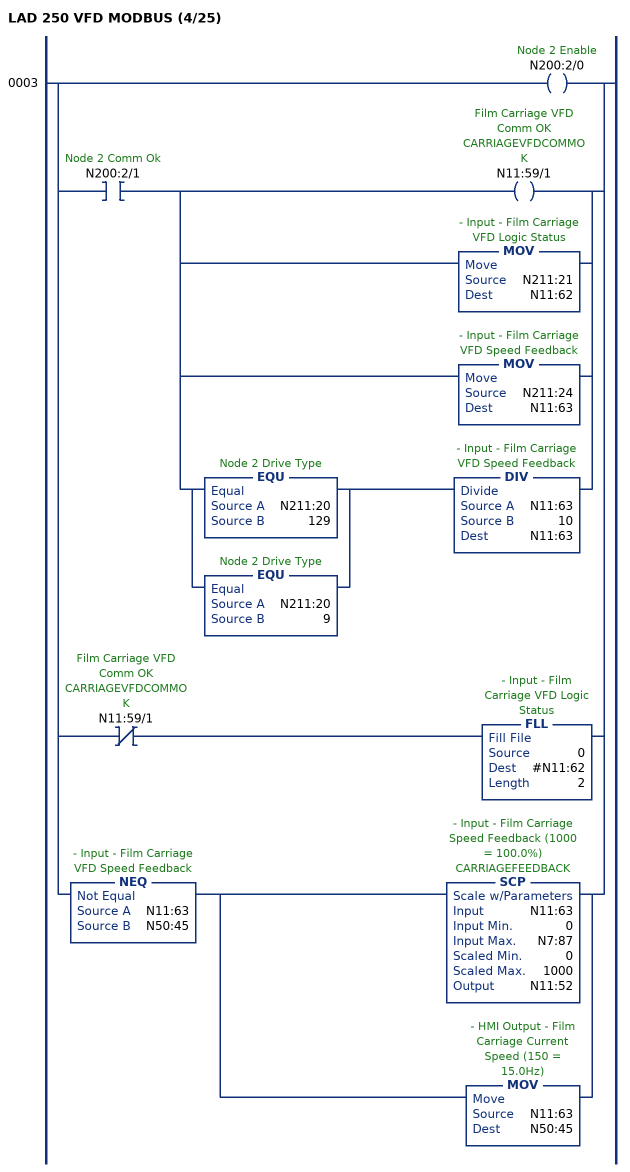
% Rung: 3 %
SOR BST OTE N200:2/0 NXB XIC N200:2/1 BST OTE N11:59/1 NXB MOV N211:21 N11:62 NXB MOV N211:24 N11:63 NXB BST EQU N211:20 129 NXB EQU N211:20 9 BND DIV N11:63 10 N11:63 BND NXB XIO N11:59/1 FLL 0 #N11:62 2 NXB NEQ N11:63 N50:45 BST SCP N11:63 0 N7:87 0 1000 N11:52 NXB MOV N11:63 N50:45 BND BND EOR
%   N200:2/0  "Node 2 Enable" %
%   N200:2/1  "Node 2 Comm Ok" %
%   N11:59/1  CARRIAGEVFDCOMMOK  "Film Carriage VFD Comm OK" %
%   N211:21  "Node 2 Logic Status" %
%   N11:62  "- Input - Film Carriage VFD Logic Status" %
%   N211:24  "Node 2 Speed Feedback" %
%   N11:63  "- Input - Film Carriage VFD Speed Feedback" %
%   N211:20  "Node 2 Drive Type" %
%   N50:45  "- HMI Output - Film Carriage Current Speed (150 = 15.0Hz)" %
%   N7:87  "Film Carriage VFD Max Hz (150 = 15.0Hz)" %
%   N11:52  CARRIAGEFEEDBACK  "- Input - Film Carriage Speed Feedback (1000 = 100.0%)" %

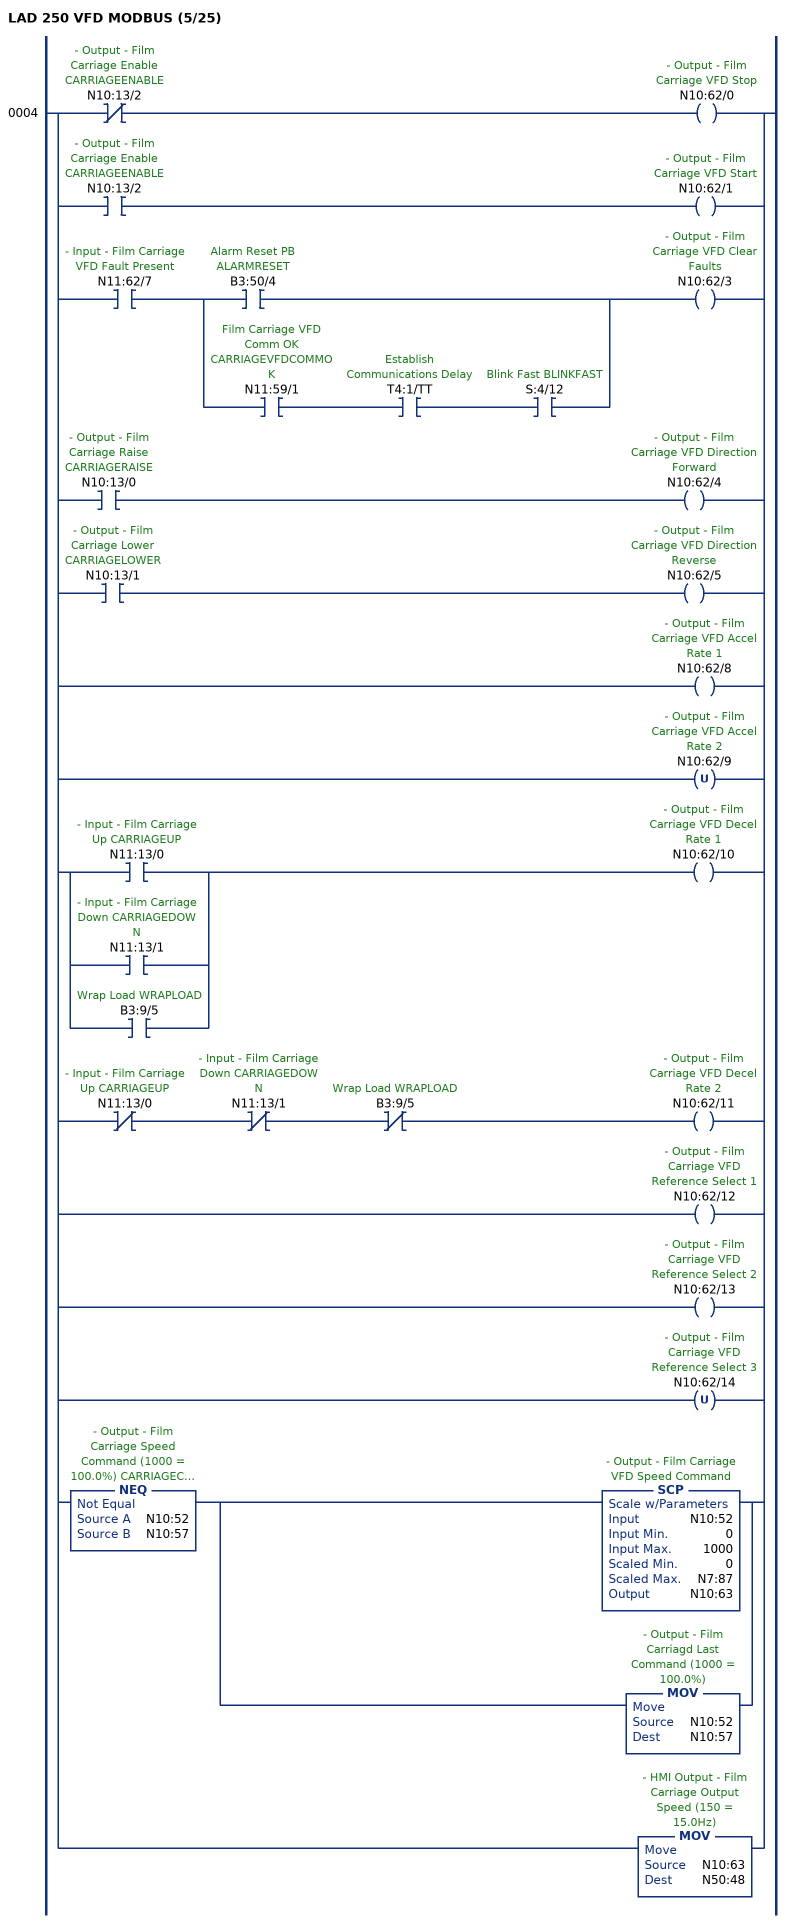
% Rung: 4 %
SOR BST XIO N10:13/2 OTE N10:62/0 NXB XIC N10:13/2 OTE N10:62/1 NXB XIC N11:62/7 BST XIC B3:50/4 NXB XIC N11:59/1 XIC T4:1/TT XIC S:4/12 BND OTE N10:62/3 NXB XIC N10:13/0 OTE N10:62/4 NXB XIC N10:13/1 OTE N10:62/5 NXB OTE N10:62/8 NXB OTU N10:62/9 NXB BST XIC N11:13/0 NXB XIC N11:13/1 NXB XIC B3:9/5 BND OTE N10:62/10 NXB XIO N11:13/0 XIO N11:13/1 XIO B3:9/5 OTE N10:62/11 NXB OTE N10:62/12 NXB OTE N10:62/13 NXB OTU N10:62/14 NXB NEQ N10:52 N10:57 BST SCP N10:52 0 1000 0 N7:87 N10:63 NXB MOV N10:52 N10:57 BND NXB MOV N10:63 N50:48 BND EOR
%   N10:13/2  CARRIAGEENABLE  "- Output - Film Carriage Enable" %
%   N10:62/0  "- Output - Film Carriage VFD Stop" %
%   N10:62/1  "- Output - Film Carriage VFD Start" %
%   N11:62/7  "- Input - Film Carriage VFD Fault Present" %
%   B3:50/4  ALARMRESET  "Alarm Reset PB" %
%   N11:59/1  CARRIAGEVFDCOMMOK  "Film Carriage VFD Comm OK" %
%   T4:1  "Establish Communications Delay" %
%   S:4/12  BLINKFAST  "Blink Fast" %
%   N10:62/3  "- Output - Film Carriage VFD Clear Faults" %
%   N10:13/0  CARRIAGERAISE  "- Output - Film Carriage Raise" %
%   N10:62/4  "- Output - Film Carriage VFD Direction Forward" %
%   N10:13/1  CARRIAGELOWER  "- Output - Film Carriage Lower" %
%   N10:62/5  "- Output - Film Carriage VFD Direction Reverse" %
%   N10:62/8  "- Output - Film Carriage VFD Accel Rate 1" %
%   N10:62/9  "- Output - Film Carriage VFD Accel Rate 2" %
%   N11:13/0  CARRIAGEUP  "- Input - Film Carriage Up" %
%   N11:13/1  CARRIAGEDOWN  "- Input - Film Carriage Down" %
%   B3:9/5  WRAPLOAD  "Wrap Load" %
%   N10:62/10  "- Output - Film Carriage VFD Decel Rate 1" %
%   N10:62/11  "- Output - Film Carriage VFD Decel Rate 2" %
%   N10:62/12  "- Output - Film Carriage VFD Reference Select 1" %
%   N10:62/13  "- Output - Film Carriage VFD Reference Select 2" %
%   N10:62/14  "- Output - Film Carriage VFD Reference Select 3" %
%   N10:52  CARRIAGECOMMAND  "- Output - Film Carriage Speed Command (1000 = 100.0%)" %
%   N10:57  "- Output - Film Carriagd Last Command (1000 = 100.0%)" %
%   N7:87  "Film Carriage VFD Max Hz (150 = 15.0Hz)" %
%   N10:63  "- Output - Film Carriage VFD Speed Command" %
%   N50:48  "- HMI Output - Film Carriage Output Speed (150 = 15.0Hz)" %

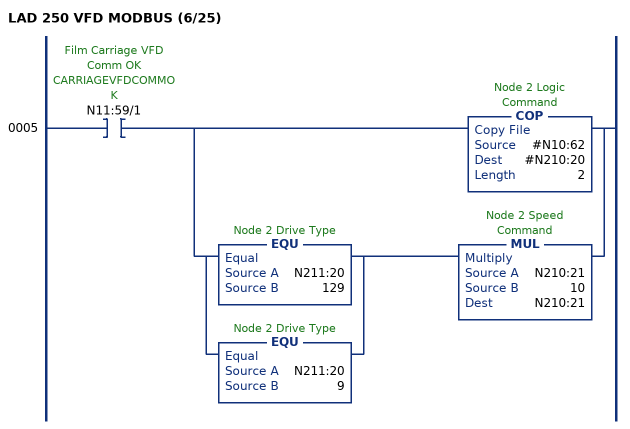
% Rung: 5 %
SOR XIC N11:59/1 BST COP #N10:62 #N210:20 2 NXB BST EQU N211:20 129 NXB EQU N211:20 9 BND MUL N210:21 10 N210:21 BND EOR
%   N11:59/1  CARRIAGEVFDCOMMOK  "Film Carriage VFD Comm OK" %
%   N10:62  "- Output - Film Carriage VFD Logic Command" %
%   N210:20  "Node 2 Logic Command" %
%   N211:20  "Node 2 Drive Type" %
%   N210:21  "Node 2 Speed Command" %

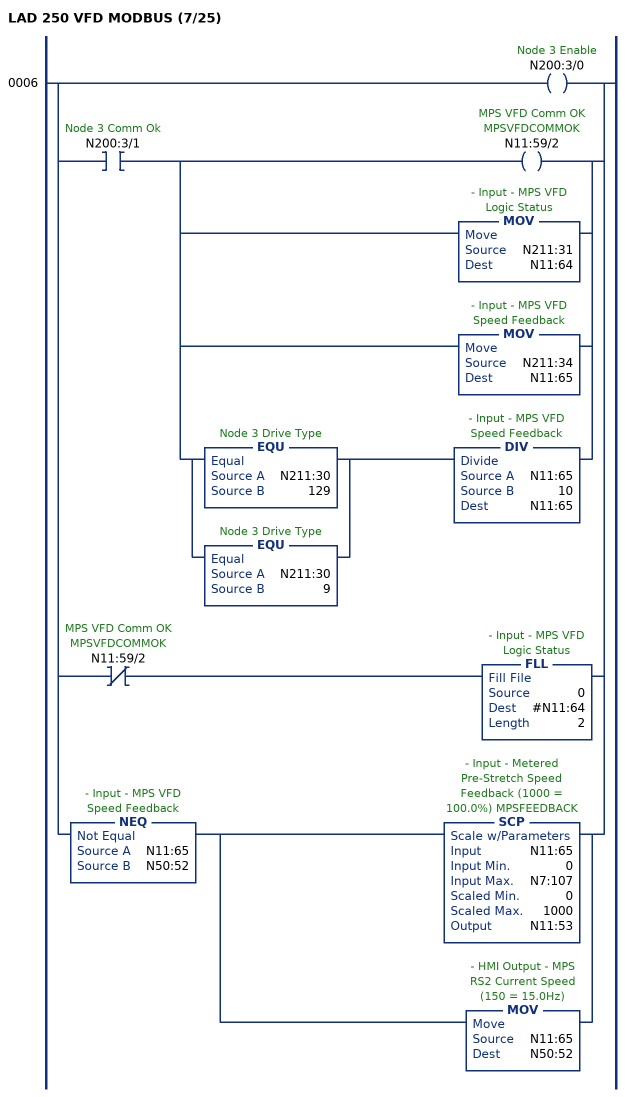
% Rung: 6 %
SOR BST OTE N200:3/0 NXB XIC N200:3/1 BST OTE N11:59/2 NXB MOV N211:31 N11:64 NXB MOV N211:34 N11:65 NXB BST EQU N211:30 129 NXB EQU N211:30 9 BND DIV N11:65 10 N11:65 BND NXB XIO N11:59/2 FLL 0 #N11:64 2 NXB NEQ N11:65 N50:52 BST SCP N11:65 0 N7:107 0 1000 N11:53 NXB MOV N11:65 N50:52 BND BND EOR
%   N200:3/0  "Node 3 Enable" %
%   N200:3/1  "Node 3 Comm Ok" %
%   N11:59/2  MPSVFDCOMMOK  "MPS VFD Comm OK" %
%   N211:31  "Node 3 Logic Status" %
%   N11:64  "- Input - MPS VFD Logic Status" %
%   N211:34  "Node 3 Speed Feedback" %
%   N11:65  "- Input - MPS VFD Speed Feedback" %
%   N211:30  "Node 3 Drive Type" %
%   N50:52  "- HMI Output - MPS RS2 Current Speed (150 = 15.0Hz)" %
%   N7:107  "Metered Pre-Stretch VFD Max Hz (150 = 15.0Hz)" %
%   N11:53  MPSFEEDBACK  "- Input - Metered Pre-Stretch Speed Feedback (1000 = 100.0%)" %

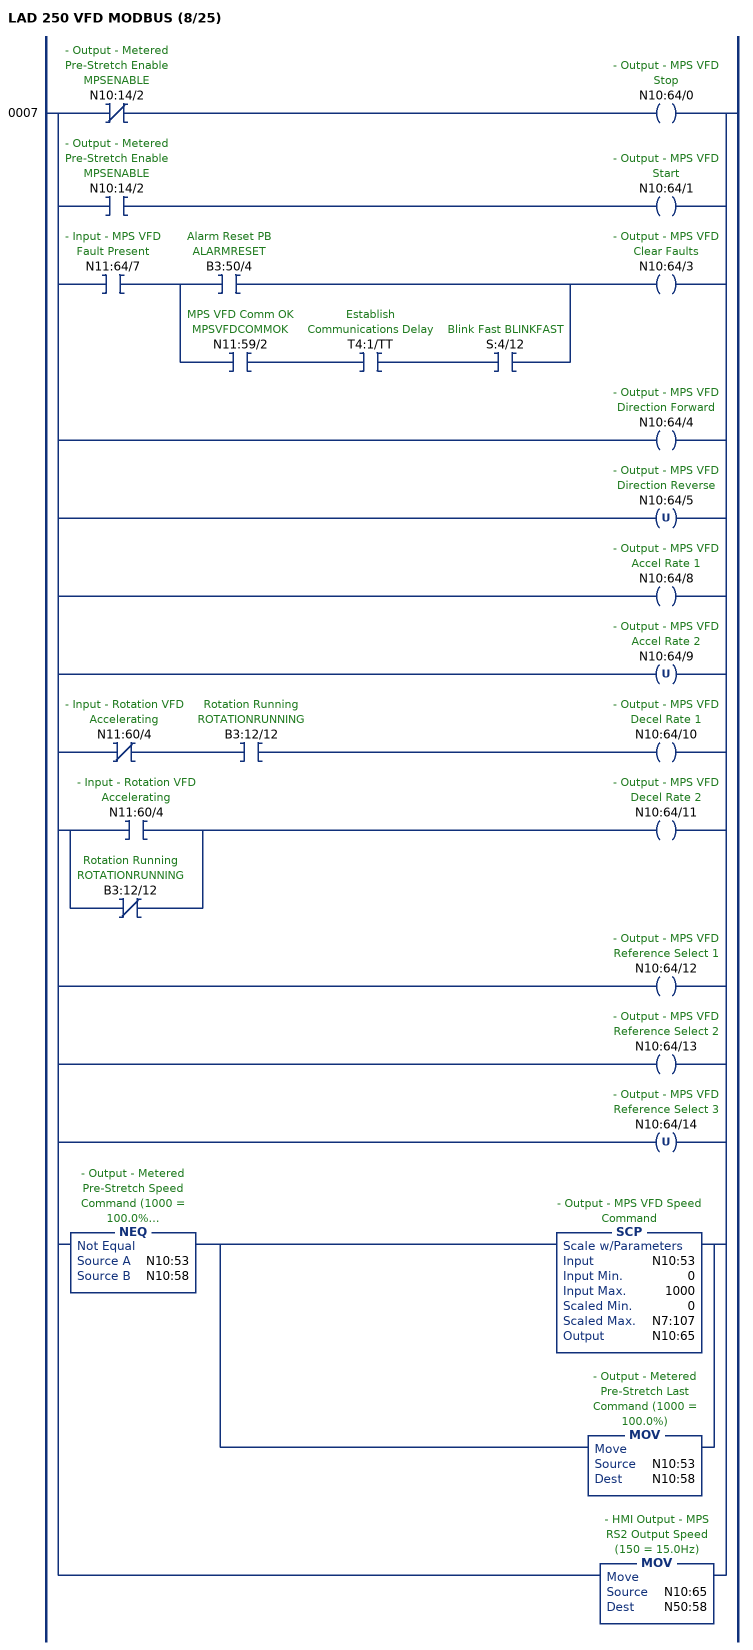
% Rung: 7 %
SOR BST XIO N10:14/2 OTE N10:64/0 NXB XIC N10:14/2 OTE N10:64/1 NXB XIC N11:64/7 BST XIC B3:50/4 NXB XIC N11:59/2 XIC T4:1/TT XIC S:4/12 BND OTE N10:64/3 NXB OTE N10:64/4 NXB OTU N10:64/5 NXB OTE N10:64/8 NXB OTU N10:64/9 NXB XIO N11:60/4 XIC B3:12/12 OTE N10:64/10 NXB BST XIC N11:60/4 NXB XIO B3:12/12 BND OTE N10:64/11 NXB OTE N10:64/12 NXB OTE N10:64/13 NXB OTU N10:64/14 NXB NEQ N10:53 N10:58 BST SCP N10:53 0 1000 0 N7:107 N10:65 NXB MOV N10:53 N10:58 BND NXB MOV N10:65 N50:58 BND EOR
%   N10:14/2  MPSENABLE  "- Output - Metered Pre-Stretch Enable" %
%   N10:64/0  "- Output - MPS VFD Stop" %
%   N10:64/1  "- Output - MPS VFD Start" %
%   N11:64/7  "- Input - MPS VFD Fault Present" %
%   B3:50/4  ALARMRESET  "Alarm Reset PB" %
%   N11:59/2  MPSVFDCOMMOK  "MPS VFD Comm OK" %
%   T4:1  "Establish Communications Delay" %
%   S:4/12  BLINKFAST  "Blink Fast" %
%   N10:64/3  "- Output - MPS VFD Clear Faults" %
%   N10:64/4  "- Output - MPS VFD Direction Forward" %
%   N10:64/5  "- Output - MPS VFD Direction Reverse" %
%   N10:64/8  "- Output - MPS VFD Accel Rate 1" %
%   N10:64/9  "- Output - MPS VFD Accel Rate 2" %
%   N11:60/4  "- Input - Rotation VFD Accelerating" %
%   B3:12/12  ROTATIONRUNNING  "Rotation Running" %
%   N10:64/10  "- Output - MPS VFD Decel Rate 1" %
%   N10:64/11  "- Output - MPS VFD Decel Rate 2" %
%   N10:64/12  "- Output - MPS VFD Reference Select 1" %
%   N10:64/13  "- Output - MPS VFD Reference Select 2" %
%   N10:64/14  "- Output - MPS VFD Reference Select 3" %
%   N10:53  MPSCOMMAND  "- Output - Metered Pre-Stretch Speed Command (1000 = 100.0%)" %
%   N10:58  "- Output - Metered Pre-Stretch Last Command (1000 = 100.0%)" %
%   N7:107  "Metered Pre-Stretch VFD Max Hz (150 = 15.0Hz)" %
%   N10:65  "- Output - MPS VFD Speed Command" %
%   N50:58  "- HMI Output - MPS RS2 Output Speed (150 = 15.0Hz)" %

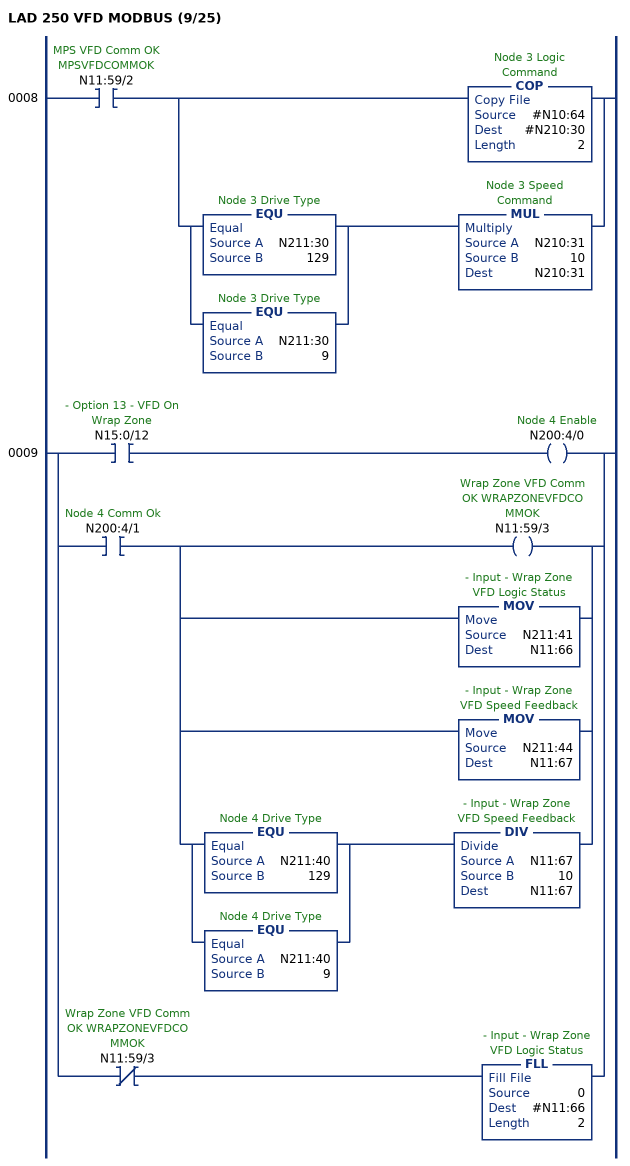
% Rung: 8 %
SOR XIC N11:59/2 BST COP #N10:64 #N210:30 2 NXB BST EQU N211:30 129 NXB EQU N211:30 9 BND MUL N210:31 10 N210:31 BND EOR
%   N11:59/2  MPSVFDCOMMOK  "MPS VFD Comm OK" %
%   N10:64  "- Output - MPS VFD Logic Command" %
%   N210:30  "Node 3 Logic Command" %
%   N211:30  "Node 3 Drive Type" %
%   N210:31  "Node 3 Speed Command" %
% Rung: 9 %
SOR BST XIC N15:0/12 OTE N200:4/0 NXB XIC N200:4/1 BST OTE N11:59/3 NXB MOV N211:41 N11:66 NXB MOV N211:44 N11:67 NXB BST EQU N211:40 129 NXB EQU N211:40 9 BND DIV N11:67 10 N11:67 BND NXB XIO N11:59/3 FLL 0 #N11:66 2 BND EOR
%   N15:0/12  "- Option 13 - VFD On Wrap Zone" %
%   N200:4/0  "Node 4 Enable" %
%   N200:4/1  "Node 4 Comm Ok" %
%   N11:59/3  WRAPZONEVFDCOMMOK  "Wrap Zone VFD Comm OK" %
%   N211:41  "Node 4 Logic Status" %
%   N11:66  "- Input - Wrap Zone VFD Logic Status" %
%   N211:44  "Node 4 Speed Feedback" %
%   N11:67  "- Input - Wrap Zone VFD Speed Feedback" %
%   N211:40  "Node 4 Drive Type" %

